(* IEC 61131-3 sources: SafeDODiag/SafeDODiag, 15 files *)

(* ---- Types.typ ---- *)
(*(Safety Release) Two-output safety contactor control and diagnosis*)
TYPE
	SContactorStateEnum :
		(
		SC_CFG := 0,
		SC_INIT,
		SC_DISABLED,
		SC_ENABLED,
		SC_ERROR := -1
		);
	SContactorCmdSimType : 	STRUCT
		EnableSim : BOOL; (*Enable contactor input and output simulation. Use fub output Simulation to see the expected output values and feedback values.*)
		SimMonitorErrors : USINT; (*Simulate error conditions by toggling individual bits to TRUE:
0: output 1 blocked by safety (interlock)
1: output 2 blocked by safety (interlock)
2: output 1 wire break (current)
3: output 2 wire break (current)
4: fdbk 1 stuck on high/"contactor open" (fdbk)
5: fdbk 2 stuck on high/"contactor open" (fdbk)
6: fdbk 1 stuck on low/"contactor closed" (fdbk)
7: fdbk 2 stuck on low/"contactor closed" (fdbk)*)
	END_STRUCT;
	SContactorCmdType : 	STRUCT
		OutputRequest : BOOL; (*Process control request: TRUE - close the contactor; FALSE - open the contactor*)
		Reset : BOOL; (*Remove the gray CPU fub from its error state and send reset request to safety CPU*)
		Simulation : SContactorCmdSimType; (*Simulation request. Element "SimMonitorErrors" only gets checked if element "EnableSim" is set to TRUE.*)
	END_STRUCT;
	SContactorCfgDiagCodeType : 	STRUCT  (*Configure safety CPU-reported SF_EDM fub DiagCode monitoring*)
		EnableMon : BOOL; (*When TRUE the contactor function block will monitor safety CPU's SF_EDM fub DiagCodes (require safety CPU to use UINT channels to pass DiagCodes to gray CPU)*)
		StartDelayTime : TIME := T#3s; (*The amount of time the gray CPU fub will delay checking SF_EDM fub DiagCode after SI card shows SafeModuleOK (must be > SF_EDM MonitorTime to allow SF_EDM to produce a stabilized DiagCode)*)
		ResetDelayTime : TIME := T#1s; (*The amount of time the gray CPU fub will delay requesting to reset SF_EDM fub after DiagCode shows 16#C060 (to allow channel diagnosis to complete and contactor feedbacks to show TRUE after SI card reports SafeModuleOK); also used as the amount of time the gray CPU fub will wait to reset itself after requesting to reset SF_EDM fub.*)
	END_STRUCT;
	SContactorCfgFdbkType : 	STRUCT  (*Configure SI hardware-based contactor status feedback monitoring*)
		EnableMon : BOOL; (*When TRUE the contactor function block will monitor SI hardware for contactor status feedback*)
		StartDelayTime : TIME := T#3s; (*The amount of time the gray CPU fub will delay checking contactor feedbacks after SI card shows SafeModuleOK (to allow channel diagnosis to complete and contactor feedbacks to show TRUE after SI card reports SafeModuleOK)*)
		MonitorTime : TIME; (*The amount of time the gray CPU fub will delay comparing contactor feedbacks to allow for switching time and debounce*)
	END_STRUCT;
	SContactorCfgCurrentType : 	STRUCT  (*Configure SO hardware-based current ok monitoring*)
		EnableMon : BOOL; (*When true the contactor function block will monitor the current input for the contactor*)
		MonitorTime : TIME; (*The amount of time the gray CPU fub will delay checking the current output to allow transient current to settle*)
	END_STRUCT;
	SContactorCfgInterlockStateType : 	STRUCT  (*Dual-channel safe digital output: Configure SO hardware-based output interlock state ("restart inhibit state") monitoring*)
		EnableMon : BOOL; (*When TRUE the contactor function block will monitor SO hardware for output interlock state (require SO card's "Restart inhibit state information" turned on)*)
		ChannelPairSelector : USINT; (*Selector for which byte of the output interlock channel represents the contactor pair (1 - contactor pair is on SO card channels 1 & 2; 3 - contactor pair is on SO card channels 3 & 4; 5 - contactor pair is on SO card channels 5 & 6; 0/2/4/etc. - selection invalid)*)
		StartDelayTime : TIME := T#3s; (*The amount of time the gray CPU fub will delay checking output interlock states after SO card shows SafeModuleOK (to allow channel diagnosis to complete after SO card reports SafeModuleOK)*)
		MonitorTime : TIME; (*The amount of time the gray CPU fub will delay comparing interlock states' discrepancy*)
	END_STRUCT;
	SContactorCfgType : 	STRUCT
		Name : STRING[35] := 'NamedContactors'; (*Unique contactor name for easy identification in alarm text*)
		DiagCode : SContactorCfgDiagCodeType; (*Option for monitoring safety CPU's SF_EDM fub state*)
		Fdbk : SContactorCfgFdbkType; (*Option for monitoring status input of each contactors*)
		Current : SContactorCfgCurrentType; (*Option for monitoring current associated with the pair of contactors*)
		InterlockState : SContactorCfgInterlockStateType; (*Option for monitoring output interlock state of each contactor*)
		BootUpDelay : TIME := T#10m; (*Wait time for the SafeModuleOK feedback on PLC startup*)
	END_STRUCT;
	SContactorSimulationType : 	STRUCT
		Input : SContactorIntInputType; (*Simulation inputs mirror the internal inputs, so the data type uses SContactorIntInputType (not a typo)*)
		Output : SContactorIntOutputType; (*Simulation inputs mirror the internal outputs, so the data type uses SContactorIntOutputType (not a typo)*)
	END_STRUCT;
	SContactorStatusType : 	STRUCT
		OutputRequested : BOOL; (*Echo the OutputRequest input to show that the fub is running*)
		OutputActive : BOOL; (*Show that both safety contactor outputs are energized (safety contactors are not necessarily closed)*)
		SafetyResetRequested : BOOL; (*Show that a SF_EDM reset needs to be sent to safety CPU*)
	END_STRUCT;
	SContactorDiagType : 	STRUCT
		DiagText : STRING[79];
		ErrorConfig : BOOL; (*The error is due to an invalid config*)
		ErrorSafeFub : BOOL; (*The error is due to safety CPU fub SF_EDM*)
		ErrorFdbk : BOOL; (*The error is due to contactor status feedback*)
		ErrorCurrent : BOOL; (*The error is due to current feedback*)
		ErrorInterlock : BOOL; (*The error is due to output interlock*)
		ErrorInternal : BOOL; (*The error is due to fub design that did not account for certain situations*)
	END_STRUCT;
	SContactorIntPrevType : 	STRUCT
		State : SContactorStateEnum;
		Reset : BOOL;
		EnDiagCode : BOOL;
		EnFdbk : BOOL;
		EnInterlock : BOOL;
		EnCurrent : BOOL;
		SimOutput1 : BOOL;
		SimOutput2 : BOOL;
	END_STRUCT;
	SContactorIntFubType : 	STRUCT
		TON_EDMStartDelay : TON;
		TON_EDMResetDelay : TON;
		TON_FdbkStartDelay : TON;
		TON_Fdbk : TON;
		TON_Current : TON;
		TON_InterlockStartDelay : TON;
		TON_Interlock : TON;
		TON_EDMMonitorSim : TON;
	END_STRUCT;
	SContactorIntInputType : 	STRUCT
		SF_In_DiagCode : UINT;
		SI_In_SafeModuleOK : BOOL;
		SI_In_Contactor1Fdbk : BOOL;
		SI_In_Contactor2Fdbk : BOOL;
		SO_In_SafeModuleOK : BOOL;
		SO_In_Output1PhysicalState : BOOL;
		SO_In_Output2PhysicalState : BOOL;
		SO_In_Output1CurrentOK : BOOL;
		SO_In_Output2CurrentOK : BOOL;
		SO_In_OutputInterlockStates : UINT;
		InterlockStateOutput1 : USINT;
		InterlockStateOutput2 : USINT;
	END_STRUCT;
	SContactorIntOutputType : 	STRUCT
		SO_Out_Contactor1 : BOOL;
		SO_Out_Contactor2 : BOOL;
	END_STRUCT;
	SContactorInternalType : 	STRUCT
		State : SContactorStateEnum; (*State of the contactor fub*)
		StateGoTo : SContactorStateEnum;
		Input : SContactorIntInputType;
		Output : SContactorIntOutputType;
		Fub : SContactorIntFubType;
		Prev : SContactorIntPrevType;
		EDMReset : BOOL;
		i : UDINT;
	END_STRUCT;
END_TYPE

(*(Safety Release) Single-channel safe digital output control and diagnosis (a simplification of SContactor)*)

TYPE
	SDigitalOutCfgInterlockStateType : 	STRUCT  (*Single-channel safe digital output: Configure SO hardware-based output interlock state ("restart inhibit state") monitoring*)
		EnableMon : BOOL; (*When TRUE the contactor function block will monitor SO hardware for output interlock state (require SO card's "Restart inhibit state information" turned on)*)
		ChannelSelector : USINT; (*Selector for which byte of the output interlock channel represents the contactor pair (1/2/3/4 for Safety Release, or 1/2 for mapp Safety - SO card channel that's being controlled; 0 or any other number - selection invalid)*)
		StartDelayTime : TIME := T#3s; (*The amount of time the gray CPU fub will delay checking output interlock states after SO card shows SafeModuleOK (to allow channel diagnosis to complete after SO card reports SafeModuleOK)*)
		MonitorTime : TIME; (*The amount of time the gray CPU fub will delay comparing interlock states' discrepancy*)
	END_STRUCT;
	SDigitalOutCfgType : 	STRUCT
		Name : STRING[35]; (*Unique contactor name for easy identification in alarm text*)
		DiagCode : SContactorCfgDiagCodeType; (*Option for monitoring safety CPU's SF_EDM fub state*)
		Fdbk : SContactorCfgFdbkType; (*Option for monitoring status input of each contactors*)
		Current : SContactorCfgCurrentType; (*Option for monitoring current associated with the pair of contactors*)
		InterlockState : SDigitalOutCfgInterlockStateType; (*Option for monitoring output interlock state of each contactor*)
	END_STRUCT;
END_TYPE

(*(mapp Safety) Interlock state monitoring for two-output safety contactor control (a modification of SContactor)*)

TYPE
	SfContactorCfgInterlockStateType : 	STRUCT  (*Dual-channel safe digital output: Configure SO hardware-based output interlock state ("error interlock state") monitoring*)
		EnableMon : BOOL; (*When TRUE the contactor function block will monitor SO hardware for output interlock state (require SO card's "Restart inhibit state information" turned on)*)
		StartDelayTime : TIME := T#3s; (*The amount of time the gray CPU fub will delay checking output interlock states after SO card shows SafeModuleOK (to allow channel diagnosis to complete after SO card reports SafeModuleOK)*)
		MonitorTime : TIME; (*The amount of time the gray CPU fub will delay comparing interlock states' discrepancy*)
	END_STRUCT;
	SfContactorCfgType : 	STRUCT
		Name : STRING[35] := 'NamedContactors'; (*Unique contactor name for easy identification in alarm text*)
		DiagCode : SContactorCfgDiagCodeType; (*Option for monitoring safety CPU's SF_EDM fub state*)
		Fdbk : SContactorCfgFdbkType; (*Option for monitoring status input of each contactors*)
		Current : SContactorCfgCurrentType; (*Option for monitoring current associated with the pair of contactors*)
		InterlockState : SfContactorCfgInterlockStateType; (*Option for monitoring output interlock state of each contactor*)
		BootUpDelay : TIME := T#10m; (*Wait time for the SafeModuleOK feedback on PLC startup*)
	END_STRUCT;
	SfContactorIntInputType : 	STRUCT
		SF_In_DiagCode : UINT;
		SI_In_SafeModuleOK : BOOL;
		SI_In_Contactor1Fdbk : BOOL;
		SI_In_Contactor2Fdbk : BOOL;
		SO_In_SafeModuleOK : BOOL;
		SO_In_Output1PhysicalState : BOOL;
		SO_In_Output2PhysicalState : BOOL;
		SO_In_Output1CurrentOK : BOOL;
		SO_In_Output2CurrentOK : BOOL;
		SO_In_OutputInterlockStates : USINT;
		InterlockStateOutput1 : USINT;
		InterlockStateOutput2 : USINT;
	END_STRUCT;
	SfContactorInternalType : 	STRUCT
		State : SContactorStateEnum; (*State of the contactor fub*)
		StateGoTo : SContactorStateEnum;
		Input : SfContactorIntInputType;
		Output : SContactorIntOutputType;
		Fub : SContactorIntFubType;
		Prev : SContactorIntPrevType;
		EDMReset : BOOL;
		i : UDINT;
	END_STRUCT;
END_TYPE

(* ---- SafeDODiag.fun ---- *)
(*Safety Release-compatible X20SO21xx/X20SO41xx output error diagnosis*)
FUNCTION_BLOCK SContactor (*Dual-channel safe digital output control and monitoring, example use includes redundant safety contactor control*)
	VAR_INPUT
		Cmd : SContactorCmdType; (*Request to energize output*)
		pSO_Out_Contactor1 : REFERENCE TO BOOL; (*Reference to the SO card output for contactor coil 1*)
		pSO_Out_Contactor2 : REFERENCE TO BOOL; (*Reference to the SO card output for contactor coil 2*)
		pSO_In_SafeModuleOK : REFERENCE TO BOOL; (*Reference to the SO card input SafeModuleOK*)
		pSO_In_Output1PhysicalState : REFERENCE TO BOOL; (*Reference to the SO card input PhysicalStateChannelX for contactor coil 1*)
		pSO_In_Output2PhysicalState : REFERENCE TO BOOL; (*Reference to the SO card input PhysicalStateChannelY for contactor coil 2*)
		Config : SContactorCfgType; (*Pointer to the configuration structure*)
		pSF_In_DiagCode : REFERENCE TO UINT; (*Reference to the safety-to-gray UINT channel that reports SF_EDM fub DiagCode*)
		pSI_In_SafeModuleOK : REFERENCE TO BOOL; (*Reference to the SO card input SafeModuleOK*)
		pSI_In_Contactor1Fdbk : REFERENCE TO BOOL; (*Reference to the SI card input for the feedback status of contactor coil 1*)
		pSI_In_Contactor2Fdbk : REFERENCE TO BOOL; (*Reference to the SI card input for the feedback status of contactor coil 2*)
		pSO_In_Output1CurrentOK : REFERENCE TO BOOL; (*Reference to the SO card's monitoring of channel current for contactor coil 1*)
		pSO_In_Output2CurrentOK : REFERENCE TO BOOL; (*Reference to the SO card's monitoring of channel current for contactor coil 2*)
		pSO_In_OutputInterlockStates : REFERENCE TO UINT; (*Reference to the SO card output interlocking states (each channel is 1 nibble in the range of 16#0 - 16#F)*)
		pSO6_In_OutputInterlockStates : REFERENCE TO UDINT; (*Reference to the SO6xxx card output interlocking states (each channel is 1 nibble in the range of 16#0 - 16#F)*)
	END_VAR
	VAR_OUTPUT
		Error : BOOL; (*Show that an error has occured to prevent output*)
		DiagCode : UINT; (*Show diagnostic code based on available monitoring capability*)
		Diag : SContactorDiagType; (*Show diagnostic info based on available monitoring capability*)
		Status : SContactorStatusType; (*Show that both safety contactor outputs are energized (safety contactors are not necessarily closed)*)
		Simulation : SContactorSimulationType; (*Show simulated I/O values based on fub input Cmd.Simulation.SimMonitorErrors*)
	END_VAR
	VAR
		Internal : SContactorInternalType; (*Internal variables*)
	END_VAR
END_FUNCTION_BLOCK

FUNCTION_BLOCK SDigitalOut (*Single-channel safe digital output control and monitoring, example use includes gas dump valve control*)
	VAR_INPUT
		Cmd : SContactorCmdType; (*Request to energize output*)
		pSO_Out_DigitalOut : REFERENCE TO BOOL; (*Reference to the SO card digital output channel*)
		pSO_In_SafeModuleOK : REFERENCE TO BOOL; (*Reference to the SO card input SafeModuleOK*)
		pSO_In_OutputPhysicalState : REFERENCE TO BOOL; (*Reference to the SO card input PhysicalStateChannelX for the controlled digital output channel*)
		Config : SDigitalOutCfgType; (*Pointer to the configuration structure*)
		pSF_In_DiagCode : REFERENCE TO UINT; (*Reference to the safety-to-gray UINT channel that reports SF_EDM fub DiagCode*)
		pSI_In_SafeModuleOK : REFERENCE TO BOOL; (*Reference to the SO card input SafeModuleOK*)
		pSI_In_DigitalOutFdbk : REFERENCE TO BOOL; (*Reference to the SI card input for the feedback status of the controlled digital output channel*)
		pSO_In_OutputCurrentOK : REFERENCE TO BOOL; (*Reference to the SO card's monitoring of channel current for the controlled digital output channel*)
		pSO_In_OutputInterlockStates : REFERENCE TO UINT; (*Reference to the SO card output interlocking states (each channel is 1 nibble in the range of 16#0 - 16#F)*)
		pSO6_In_OutputInterlockStates : REFERENCE TO UDINT; (*Reference to the SO6xxx card output interlocking states (each channel is 1 nibble in the range of 16#0 - 16#F)*)
	END_VAR
	VAR_OUTPUT
		Error : BOOL; (*Show that an error has occured to prevent output*)
		DiagCode : UINT; (*Show diagnostic code based on available monitoring capability*)
		Diag : SContactorDiagType; (*Show diagnostic info based on available monitoring capability*)
		Status : SContactorStatusType; (*Show that safety digiral output is energized*)
		Simulation : SContactorSimulationType; (*Show simulated I/O values based on fub input Cmd.Simulation.SimMonitorErrors*)
	END_VAR
	VAR
		Internal : SContactorInternalType; (*Internal variables*)
	END_VAR
END_FUNCTION_BLOCK
(*mapp Safety-compatible X20SO21xx/X20SO41xx output error diagnosis*)

FUNCTION_BLOCK SfContactor (*Dual-channel safe digital output control and monitoring, example use includes redundant safety contactor control*)
	VAR_INPUT
		Cmd : SContactorCmdType; (*Request to energize output*)
		pSO_Out_Contactor1 : REFERENCE TO BOOL; (*Reference to the SO card output for contactor coil 1*)
		pSO_Out_Contactor2 : REFERENCE TO BOOL; (*Reference to the SO card output for contactor coil 2*)
		pSO_In_SafeModuleOK : REFERENCE TO BOOL; (*Reference to the SO card input SafeModuleOK*)
		pSO_In_Output1PhysicalState : REFERENCE TO BOOL; (*Reference to the SO card input PhysicalStateChannelX for contactor coil 1*)
		pSO_In_Output2PhysicalState : REFERENCE TO BOOL; (*Reference to the SO card input PhysicalStateChannelY for contactor coil 2*)
		Config : SfContactorCfgType; (*Pointer to the configuration structure*)
		pSF_In_DiagCode : REFERENCE TO UINT; (*Reference to the safety-to-gray UINT channel that reports SF_EDM fub DiagCode*)
		pSI_In_SafeModuleOK : REFERENCE TO BOOL; (*Reference to the SO card input SafeModuleOK*)
		pSI_In_Contactor1Fdbk : REFERENCE TO BOOL; (*Reference to the SI card input for the feedback status of contactor coil 1*)
		pSI_In_Contactor2Fdbk : REFERENCE TO BOOL; (*Reference to the SI card input for the feedback status of contactor coil 2*)
		pSO_In_Output1CurrentOK : REFERENCE TO BOOL; (*Reference to the SO card's monitoring of channel current for contactor coil 1*)
		pSO_In_Output2CurrentOK : REFERENCE TO BOOL; (*Reference to the SO card's monitoring of channel current for contactor coil 2*)
		pSO_In_OutputInterlockStates : REFERENCE TO USINT; (*Reference to the SO card output interlocking states (each channel is 1 nibble in the range of 16#0 - 16#F)*)
	END_VAR
	VAR_OUTPUT
		Error : BOOL; (*Show that an error has occured to prevent output*)
		DiagCode : UINT; (*Show diagnostic code based on available monitoring capability*)
		Diag : SContactorDiagType; (*Show diagnostic info based on available monitoring capability*)
		Status : SContactorStatusType; (*Show that both safety contactor outputs are energized (safety contactors are not necessarily closed)*)
		Simulation : SContactorSimulationType; (*Show simulated I/O values based on fub input Cmd.Simulation.SimMonitorErrors*)
	END_VAR
	VAR
		Internal : SfContactorInternalType; (*Internal variables*)
	END_VAR
END_FUNCTION_BLOCK

FUNCTION_BLOCK SfDigitalOut (*Single-channel safe digital output control and monitoring, example use includes gas dump valve control*)
	VAR_INPUT
		Cmd : SContactorCmdType; (*Request to energize output*)
		pSO_Out_DigitalOut : REFERENCE TO BOOL; (*Reference to the SO card digital output channel*)
		pSO_In_SafeModuleOK : REFERENCE TO BOOL; (*Reference to the SO card input SafeModuleOK*)
		pSO_In_OutputPhysicalState : REFERENCE TO BOOL; (*Reference to the SO card input PhysicalStateChannelX for the controlled digital output channel*)
		Config : SDigitalOutCfgType; (*Pointer to the configuration structure*)
		pSF_In_DiagCode : REFERENCE TO UINT; (*Reference to the safety-to-gray UINT channel that reports SF_EDM fub DiagCode*)
		pSI_In_SafeModuleOK : REFERENCE TO BOOL; (*Reference to the SO card input SafeModuleOK*)
		pSI_In_DigitalOutFdbk : REFERENCE TO BOOL; (*Reference to the SI card input for the feedback status of the controlled digital output channel*)
		pSO_In_OutputCurrentOK : REFERENCE TO BOOL; (*Reference to the SO card's monitoring of channel current for the controlled digital output channel*)
		pSO_In_OutputInterlockStates : REFERENCE TO USINT; (*Reference to the SO card output interlocking states (each channel is 1 nibble in the range of 16#0 - 16#F)*)
	END_VAR
	VAR_OUTPUT
		Error : BOOL; (*Show that an error has occured to prevent output*)
		DiagCode : UINT; (*Show diagnostic code based on available monitoring capability*)
		Diag : SContactorDiagType; (*Show diagnostic info based on available monitoring capability*)
		Status : SContactorStatusType; (*Show that safety digiral output is energized*)
		Simulation : SContactorSimulationType; (*Show simulated I/O values based on fub input Cmd.Simulation.SimMonitorErrors*)
	END_VAR
	VAR
		Internal : SfContactorInternalType; (*Internal variables*)
	END_VAR
END_FUNCTION_BLOCK

(* ---- SContactor.st ---- *)
(*
This fub has four monitoring options, ordered by priority below:
1) SF_EDM DiagCode from safety CPU (highest priority)
2) external contactor state monitoring (using SafeDigitalInput0x from SI card)
3) internal contactor wiring monitoring (using CurrentOK0x from SO card)
4) output interlock state monitoring (using FBK_Status_1 from SO card) (lowest priority)
If more than one monitoring options are enabled, the highest priority option will be used by the fub to evaluate contactor open/close behavior.
##################################################*)

FUNCTION_BLOCK SContactor

	//########## Simulation input handling ##########
	IF ( Cmd.Simulation.EnableSim ) THEN
		Simulation.Input.SI_In_SafeModuleOK	:= TRUE;
		Simulation.Input.SO_In_SafeModuleOK	:= TRUE;

		Internal.i	:= TIME_TO_UDINT( clock_ms() ) MOD 200;

		//########## SContactor dual-channel input simulation ##########
		// SimMonitorErrors bits (when set to TRUE):
		//  0: output 1 blocked by safety (interlock)
		//  1: output 2 blocked by safety (interlock)
		//  2: output 1 wire break (current)
		//  3: output 2 wire break (current)
		//  4: fdbk 1 stuck on high/"contactor open" (fdbk)
		//  5: fdbk 2 stuck on high/"contactor open" (fdbk)
		//  6: fdbk 1 stuck on low/"contactor closed" (fdbk)
		//  7: fdbk 2 stuck on low/"contactor closed" (fdbk)

		// simulate interlock feedback
		IF ( Cmd.Simulation.SimMonitorErrors.0 ) THEN
			Simulation.Input.SO_In_Output1PhysicalState	:= FALSE;
			Simulation.Input.InterlockStateOutput1		:= 8;
		ELSE
			Simulation.Input.SO_In_Output1PhysicalState	:= Simulation.Output.SO_Out_Contactor1 AND ( Simulation.Input.SO_In_Output1PhysicalState OR ( Internal.i >= 0	AND Internal.i < 50 ) );
			IF ( Simulation.Input.SO_In_Output1PhysicalState ) THEN
				Simulation.Input.InterlockStateOutput1	:= 9;
			ELSE
				Simulation.Input.InterlockStateOutput1	:= 7;
			END_IF
		END_IF
		IF ( Cmd.Simulation.SimMonitorErrors.1 ) THEN
			Simulation.Input.SO_In_Output2PhysicalState	:= FALSE;
			Simulation.Input.InterlockStateOutput2		:= 8;
		ELSE
			Simulation.Input.SO_In_Output2PhysicalState	:= Simulation.Output.SO_Out_Contactor2 AND ( Simulation.Input.SO_In_Output2PhysicalState OR ( Internal.i >= 15	AND Internal.i < 65 ) );
			IF ( Simulation.Input.SO_In_Output2PhysicalState ) THEN
				Simulation.Input.InterlockStateOutput2	:= 9;
			ELSE
				Simulation.Input.InterlockStateOutput2	:= 7;
			END_IF
		END_IF

		// simulate current ok feedback
		IF ( Cmd.Simulation.SimMonitorErrors.2 ) THEN
			Simulation.Input.SO_In_Output1CurrentOK	:= FALSE;
		ELSE
			Simulation.Input.SO_In_Output1CurrentOK	:= Simulation.Input.SO_In_Output1PhysicalState AND ( Simulation.Input.SO_In_Output1CurrentOK OR ( Internal.i >= 30	AND Internal.i < 80 ) );
		END_IF
		IF ( Cmd.Simulation.SimMonitorErrors.3 ) THEN
			Simulation.Input.SO_In_Output2CurrentOK	:= FALSE;
		ELSE
			Simulation.Input.SO_In_Output2CurrentOK	:= Simulation.Input.SO_In_Output2PhysicalState AND ( Simulation.Input.SO_In_Output2CurrentOK OR ( Internal.i >= 45	AND Internal.i < 95 ) );
		END_IF

		// simulate external monitoring feedback
		IF ( Cmd.Simulation.SimMonitorErrors.4 ) THEN
			Simulation.Input.SI_In_Contactor1Fdbk	:= TRUE;
		ELSIF ( Cmd.Simulation.SimMonitorErrors.6 ) THEN
			Simulation.Input.SI_In_Contactor1Fdbk	:= FALSE;
		ELSE
			IF ( Internal.i >= 60 AND Internal.i < 110 ) THEN
				IF ( Simulation.Input.SO_In_Output1CurrentOK ) THEN
					Simulation.Input.SI_In_Contactor1Fdbk	:= FALSE;
				ELSE
					Simulation.Input.SI_In_Contactor1Fdbk	:= TRUE;
				END_IF
			END_IF
		END_IF
		IF ( Cmd.Simulation.SimMonitorErrors.5 ) THEN
			Simulation.Input.SI_In_Contactor2Fdbk	:= TRUE;
		ELSIF ( Cmd.Simulation.SimMonitorErrors.7 ) THEN
			Simulation.Input.SI_In_Contactor2Fdbk	:= FALSE;
		ELSE
			IF ( Internal.i >= 75 AND Internal.i < 125 ) THEN
				IF ( Simulation.Input.SO_In_Output2CurrentOK ) THEN
					Simulation.Input.SI_In_Contactor2Fdbk	:= FALSE;
				ELSE
					Simulation.Input.SI_In_Contactor2Fdbk	:= TRUE;
				END_IF
			END_IF
		END_IF

		//########## DiagCode simulation ##########
		SimAction_DiagCode;

		//########## SContactor dual-channel input source assignment ##########
		Internal.Input.SF_In_DiagCode		:= Simulation.Input.SF_In_DiagCode;
		Internal.Input.SI_In_SafeModuleOK		:= Simulation.Input.SI_In_SafeModuleOK;
		Internal.Input.SI_In_Contactor1Fdbk		:= Simulation.Input.SI_In_Contactor1Fdbk;
		Internal.Input.SI_In_Contactor2Fdbk		:= Simulation.Input.SI_In_Contactor2Fdbk;
		Internal.Input.SO_In_SafeModuleOK			:= Simulation.Input.SO_In_SafeModuleOK;
		Internal.Input.SO_In_Output1PhysicalState	:= Simulation.Input.SO_In_Output1PhysicalState;
		Internal.Input.SO_In_Output2PhysicalState	:= Simulation.Input.SO_In_Output2PhysicalState;
		Internal.Input.SO_In_Output1CurrentOK		:= Simulation.Input.SO_In_Output1CurrentOK;
		Internal.Input.SO_In_Output2CurrentOK		:= Simulation.Input.SO_In_Output2CurrentOK;
		IF ( Config.InterlockState.ChannelPairSelector = 1 ) THEN
			Internal.Input.SO_In_OutputInterlockStates	:= Simulation.Input.InterlockStateOutput1 + Simulation.Input.InterlockStateOutput2 * 16#10;
		ELSIF ( Config.InterlockState.ChannelPairSelector = 3 ) THEN
			Internal.Input.SO_In_OutputInterlockStates	:= Simulation.Input.InterlockStateOutput1 * 16#100 + Simulation.Input.InterlockStateOutput2 * 16#1000;
		ELSIF ( Config.InterlockState.ChannelPairSelector = 5 AND ADR(pSO6_In_OutputInterlockStates) > 0 ) THEN
			Internal.Input.SO_In_OutputInterlockStates	:= Simulation.Input.InterlockStateOutput1 * 16#10000 + Simulation.Input.InterlockStateOutput2 * 16#100000;
		ELSE
			Internal.Input.SO_In_OutputInterlockStates	:= 0;
		END_IF

	ELSE
		//########## SContactor dual-channel input source assignment ##########
		IF ( ADR(pSF_In_DiagCode) > 0 ) THEN
			Internal.Input.SF_In_DiagCode		:= pSF_In_DiagCode;
		ELSE
			Internal.Input.SF_In_DiagCode		:= 0;
		END_IF
		IF ( ADR(pSI_In_SafeModuleOK) > 0 ) THEN
			Internal.Input.SI_In_SafeModuleOK	:= pSI_In_SafeModuleOK;
		ELSE
			Internal.Input.SI_In_SafeModuleOK	:= 0;
		END_IF
		IF ( ADR(pSI_In_Contactor1Fdbk) > 0 ) THEN
			Internal.Input.SI_In_Contactor1Fdbk	:= pSI_In_Contactor1Fdbk;
		ELSE
			Internal.Input.SI_In_Contactor1Fdbk	:= 0;
		END_IF
		IF ( ADR(pSI_In_Contactor2Fdbk) > 0 ) THEN
			Internal.Input.SI_In_Contactor2Fdbk	:= pSI_In_Contactor2Fdbk;
		ELSE
			Internal.Input.SI_In_Contactor2Fdbk	:= 0;
		END_IF
		IF ( ADR(pSO_In_SafeModuleOK) > 0 ) THEN
			Internal.Input.SO_In_SafeModuleOK			:= pSO_In_SafeModuleOK;
		ELSE
			Internal.Input.SO_In_SafeModuleOK			:= 0;
		END_IF
		IF ( ADR(pSO_In_Output1PhysicalState) > 0 ) THEN
			Internal.Input.SO_In_Output1PhysicalState	:= pSO_In_Output1PhysicalState;
		ELSE
			Internal.Input.SO_In_Output1PhysicalState	:= 0;
		END_IF
		IF ( ADR(pSO_In_Output2PhysicalState) > 0 ) THEN
			Internal.Input.SO_In_Output2PhysicalState	:= pSO_In_Output2PhysicalState;
		ELSE
			Internal.Input.SO_In_Output2PhysicalState	:= 0;
		END_IF
		IF ( ADR(pSO_In_Output1CurrentOK) > 0 ) THEN
			Internal.Input.SO_In_Output1CurrentOK		:= pSO_In_Output1CurrentOK;
		ELSE
			Internal.Input.SO_In_Output1CurrentOK		:= 0;
		END_IF
		IF ( ADR(pSO_In_Output2CurrentOK) > 0 ) THEN
			Internal.Input.SO_In_Output2CurrentOK		:= pSO_In_Output2CurrentOK;
		ELSE
			Internal.Input.SO_In_Output2CurrentOK		:= 0;
		END_IF
		IF ( ADR(pSO6_In_OutputInterlockStates) > 0 ) THEN
			Internal.Input.SO_In_OutputInterlockStates	:= pSO6_In_OutputInterlockStates;
		ELSIF ( ADR(pSO_In_OutputInterlockStates) > 0 ) THEN
			Internal.Input.SO_In_OutputInterlockStates	:= UINT_TO_UDINT( pSO_In_OutputInterlockStates );
		ELSE
			Internal.Input.SO_In_OutputInterlockStates	:= 0;
		END_IF
		//########## Reset simulation inputs ##########
		brsmemset( ADR(Simulation.Input), 0, SIZEOF(Simulation.Input) );

	END_IF

	//########## SContactor dual-channel output interlock state identification ##########
	// Read output channel interlock state
	IF ( Config.InterlockState.EnableMon ) THEN
		CASE Config.InterlockState.ChannelPairSelector OF
			1:
				Internal.Input.InterlockStateOutput1 := UDINT_TO_USINT( Internal.Input.SO_In_OutputInterlockStates AND 16#00000F );
				Internal.Input.InterlockStateOutput2 := UDINT_TO_USINT( SHR(( Internal.Input.SO_In_OutputInterlockStates AND 16#0000F0 ), 4) );
			3:
				Internal.Input.InterlockStateOutput1 := UDINT_TO_USINT( SHR(( Internal.Input.SO_In_OutputInterlockStates AND 16#000F00 ), 8) );
				Internal.Input.InterlockStateOutput2 := UDINT_TO_USINT( SHR(( Internal.Input.SO_In_OutputInterlockStates AND 16#00F000 ), 12) );
			5:
				IF ( ADR(pSO6_In_OutputInterlockStates) > 0 ) THEN
					Internal.Input.InterlockStateOutput1 := UDINT_TO_USINT( SHR(( Internal.Input.SO_In_OutputInterlockStates AND 16#0F0000 ), 16) );
					Internal.Input.InterlockStateOutput2 := UDINT_TO_USINT( SHR(( Internal.Input.SO_In_OutputInterlockStates AND 16#F00000 ), 20) );
				ELSE
					Internal.Input.InterlockStateOutput1 := 0;
					Internal.Input.InterlockStateOutput2 := 0;
				END_IF
			ELSE
				Internal.Input.InterlockStateOutput1 := 0;
				Internal.Input.InterlockStateOutput2 := 0;
		END_CASE
	ELSE
		Internal.Input.InterlockStateOutput1 := 0;
		Internal.Input.InterlockStateOutput2 := 0;
	END_IF

	//########## Feedback interpretation and error state transition ##########
	StateAction_CommonPre;

	//########## State machine for processing feedback values ##########
	CASE Internal.State OF

		SC_CFG:
			//#################### Req. Checkout ####################
			IF ( ADR(pSO_In_SafeModuleOK) = 0 ) THEN // Check if the monitoring of safe communication to SO node exists
				DiagCode			:= 16#F001;
				Diag.ErrorConfig	:= TRUE;
				Diag.DiagText		:= 'NoSafeDOCardOkADR';
			ELSIF ( ADR(pSO_Out_Contactor1) = 0 ) THEN // Check if output channe l exists
				DiagCode			:= 16#F002;
				Diag.ErrorConfig	:= TRUE;
				Diag.DiagText		:= 'NoContactor1OutADR';
			ELSIF ( ADR(pSO_Out_Contactor2) = 0 ) THEN // Check if output channe 2 exists
				DiagCode			:= 16#F003;
				Diag.ErrorConfig	:= TRUE;
				Diag.DiagText		:= 'NoContactor2OutADR';
			ELSIF ( ADR(pSO_In_Output1PhysicalState) = 0 ) THEN // Check if the output phsical state monitoring exists
				DiagCode			:= 16#F004;
				Diag.ErrorConfig	:= TRUE;
				Diag.DiagText		:= 'NoOutput1PhysicalStateADR';
			ELSIF ( ADR(pSO_In_Output2PhysicalState) = 0 ) THEN // Check if the output phsical state monitoring exists
				DiagCode			:= 16#F005;
				Diag.ErrorConfig	:= TRUE;
				Diag.DiagText		:= 'NoOutput2PhysicalStateADR';
			END_IF
			// No MonitorTime for PhysicalState because we don't know when the safety CPU will approve output enable request

			//#################### Check the setup of safety-to-gray comm of SF_EDM fub DiagCode monitor ##################
			IF ( Config.DiagCode.EnableMon AND NOT(Diag.ErrorConfig) ) THEN
				IF ( ADR(pSF_In_DiagCode) = 0 ) THEN // Check if the monitoring of DiagCode from safety CPU exists
					DiagCode			:= 16#F010;
					Diag.ErrorConfig	:= TRUE;
					Diag.DiagText		:= 'NoDiagCodeADR';
				ELSIF ( ADR(pSI_In_SafeModuleOK) = 0 ) THEN // Check if the monitoring of safe communication to SI node exists
					DiagCode			:= 16#F011;
					Diag.ErrorConfig	:= TRUE;
					Diag.DiagText		:= 'NoSafeDICardOkADR';
				ELSIF ( ADR(pSI_In_Contactor1Fdbk) = 0 ) THEN // Need an SI card input to monitor
					DiagCode			:= 16#F012;
					Diag.ErrorConfig	:= TRUE;
					Diag.DiagText		:= 'NoContactor1FdbkADR';
				ELSIF ( ADR(pSI_In_Contactor2Fdbk) = 0 ) THEN // Need an SI card input to monitor
					DiagCode			:= 16#F013;
					Diag.ErrorConfig	:= TRUE;
					Diag.DiagText		:= 'NoContactor2FdbkADR';
				ELSIF ( Config.DiagCode.StartDelayTime = 0 ) THEN // Check time range
					DiagCode			:= 16#F020;
					Diag.ErrorConfig	:= TRUE;
					Diag.DiagText		:= 'NoStartDelay';
				ELSIF ( Config.DiagCode.StartDelayTime > T#2m ) THEN // Check time range
					DiagCode			:= 16#F021;
					Diag.ErrorConfig	:= TRUE;
					Diag.DiagText		:= 'StartDelayTooLong';
				ELSIF ( Config.DiagCode.ResetDelayTime = 0 ) THEN // Check time range
					DiagCode			:= 16#F022;
					Diag.ErrorConfig	:= TRUE;
					Diag.DiagText		:= 'NoResetDelay';
				ELSIF ( Config.DiagCode.ResetDelayTime > T#10s ) THEN // Check time range
					DiagCode			:= 16#F023;
					Diag.ErrorConfig	:= TRUE;
					Diag.DiagText		:= 'ResetDelayTooLong';
				END_IF

			//#################### Check the setup of Contactor Feedback monitor ####################
			ELSIF ( Config.Fdbk.EnableMon AND NOT(Diag.ErrorConfig) ) THEN
				IF ( ADR(pSI_In_SafeModuleOK) = 0 ) THEN // Check if the monitoring of safe communication to SI node exists
					DiagCode			:= 16#F011;
					Diag.ErrorConfig	:= TRUE;
					Diag.DiagText		:= 'NoSafeDICardOkADR';
				ELSIF ( ADR(pSI_In_Contactor1Fdbk) = 0 ) THEN // Need an SI card input to monitor
					DiagCode			:= 16#F012;
					Diag.ErrorConfig	:= TRUE;
					Diag.DiagText		:= 'NoContactor1FdbkADR';
				ELSIF ( ADR(pSI_In_Contactor2Fdbk) = 0 ) THEN // Need an SI card input to monitor
					DiagCode			:= 16#F013;
					Diag.ErrorConfig	:= TRUE;
					Diag.DiagText		:= 'NoContactor2FdbkADR';
				ELSIF ( Config.Fdbk.StartDelayTime = 0 ) THEN // Check time range
					DiagCode			:= 16#F020;
					Diag.ErrorConfig	:= TRUE;
					Diag.DiagText		:= 'NoStartDelay';
				ELSIF ( Config.Fdbk.StartDelayTime > T#10s ) THEN // Check time range
					DiagCode			:= 16#F021;
					Diag.ErrorConfig	:= TRUE;
					Diag.DiagText		:= 'StartDelayTooLong';
				ELSIF ( Config.Fdbk.MonitorTime = 0 ) THEN // Check time range
					DiagCode			:= 16#F024;
					Diag.ErrorConfig	:= TRUE;
					Diag.DiagText		:= 'NoMonitorTime';
				ELSIF ( Config.Fdbk.MonitorTime > T#2s ) THEN // Check time range
					DiagCode			:= 16#F025;
					Diag.ErrorConfig	:= TRUE;
					Diag.DiagText		:= 'MonitorTimeTooLong';
				END_IF

			//#################### Check the setup of Output Current monitor ##################
			ELSIF ( Config.Current.EnableMon AND NOT(Diag.ErrorConfig) ) THEN
				IF ( ADR(pSO_In_Output1CurrentOK) = 0 ) THEN
					DiagCode			:= 16#F014;
					Diag.ErrorConfig	:= TRUE;
					Diag.DiagText		:= 'NoOutput1CurrentOkADR';
				ELSIF ( ADR(pSO_In_Output2CurrentOK) = 0 ) THEN
					DiagCode			:= 16#F015;
					Diag.ErrorConfig	:= TRUE;
					Diag.DiagText		:= 'NoOutput2CurrentOkADR';
				ELSIF ( Config.Current.MonitorTime = 0 ) THEN // Check time range
					DiagCode			:= 16#F024;
					Diag.ErrorConfig	:= TRUE;
					Diag.DiagText		:= 'NoMonitorTime';
				ELSIF ( Config.Current.MonitorTime > T#2s ) THEN // Check time range
					DiagCode			:= 16#F025;
					Diag.ErrorConfig	:= TRUE;
					Diag.DiagText		:= 'MonitorTimeTooLong';
				END_IF

			//#################### Check the setup of Output Interlock monitor ##################
			ELSIF ( Config.InterlockState.EnableMon AND NOT(Diag.ErrorConfig) ) THEN
				IF ( ( ADR(pSO_In_OutputInterlockStates) = 0 AND ADR(pSO6_In_OutputInterlockStates) = 0 )
					OR ( Config.InterlockState.ChannelPairSelector = 5 AND ADR(pSO6_In_OutputInterlockStates) = 0 )
					) THEN
					DiagCode			:= 16#F016;
					Diag.ErrorConfig	:= TRUE;
					Diag.DiagText		:= 'NoOutputInterlockStateADR';
				ELSIF ( Config.InterlockState.MonitorTime = 0 ) THEN // Check time range
					DiagCode			:= 16#F024;
					Diag.ErrorConfig	:= TRUE;
					Diag.DiagText		:= 'NoMonitorTime';
				ELSIF ( Config.InterlockState.MonitorTime > T#1s ) THEN // Check time range
					DiagCode			:= 16#F025;
					Diag.ErrorConfig	:= TRUE;
					Diag.DiagText		:= 'MonitorTimeTooLong';
				ELSIF ( (Config.InterlockState.ChannelPairSelector <> 1)
					AND (Config.InterlockState.ChannelPairSelector <> 3)
					AND (Config.InterlockState.ChannelPairSelector <> 5)
					) THEN
					DiagCode			:= 16#F026;
					Diag.ErrorConfig	:= TRUE;
					Diag.DiagText		:= 'InvalidOutputInterlockChannelPairSelector';
				END_IF
			END_IF

			//#################### SUCCESS!!! ##################
			IF NOT( Diag.ErrorConfig ) THEN
				Internal.StateGoTo	:= SC_INIT;
			END_IF

		SC_INIT:
			StateAction_Init;

		SC_DISABLED:
			StateAction_Disabled;

		SC_ENABLED:
			StateAction_Enabled;

		SC_ERROR:
			StateAction_Error;

		ELSE
			//The code should not end uzp here. Report the error as unknown.
			Diag.ErrorInternal	:= TRUE;
			DiagCode			:= 16#CFFF;
			Diag.DiagText		:= 'UndocumentedError';

	END_CASE

	//########## Update fub outputs ##########
	// Update fub error output
	Error := Diag.ErrorSafeFub OR Diag.ErrorInterlock OR Diag.ErrorCurrent OR Diag.ErrorFdbk OR Diag.ErrorConfig OR Diag.ErrorInternal;

	// Update fub IO status outputs
	IF ( Internal.State > SC_INIT ) THEN
		// Update IOSP outputs after fub init is successful, so all safety outputs are in a safe state before energizing and monitoring
		Internal.Output.SO_Out_Contactor1	:= Cmd.OutputRequest;
		Internal.Output.SO_Out_Contactor2	:= Cmd.OutputRequest;

		// Update fub status outputs based on IOSP dual-channel agreement
		Status.OutputActive		:= Internal.Input.SO_In_Output1PhysicalState AND Internal.Input.SO_In_Output2PhysicalState; // both channels need to activate to energize, so all dual-channel diagreements are treated as inactive
		Status.OutputRequested	:= Internal.Output.SO_Out_Contactor1 AND Internal.Output.SO_Out_Contactor2; // both channels need to activate to energize, so all dual-channel diagreements are treated as no request
	ELSE
		// disable IOSP output during CFG state or ERROR state
		Internal.Output.SO_Out_Contactor1	:= FALSE;
		Internal.Output.SO_Out_Contactor2	:= FALSE;

		// Update fub status output based on available SContactor dual-channel IOSP data
		IF ( ADR(pSO_In_Output1PhysicalState) > 0 AND ADR(pSO_In_Output2PhysicalState) > 0 ) THEN
			Status.OutputActive	:= Internal.Input.SO_In_Output1PhysicalState AND Internal.Input.SO_In_Output2PhysicalState;
		ELSIF ( ADR(pSO_In_Output1PhysicalState) > 0 ) THEN
			Status.OutputActive	:= Internal.Input.SO_In_Output1PhysicalState;
		ELSIF ( ADR(pSO_In_Output2PhysicalState) > 0 ) THEN
			Status.OutputActive	:= Internal.Input.SO_In_Output2PhysicalState;
		ELSE
			Status.OutputActive	:= FALSE;
		END_IF
		Status.OutputRequested	:= FALSE;
	END_IF

	// Disable internal EDM reset request after a jump out of init state that's not made within the state machine (presumably into error state)
	// Note: Error state sets internal EDM reset request on rising edge of error acknowledgement, so error state needs to disable EDM reset on its own
	IF ( Internal.Prev.State = SC_INIT AND Internal.State <> SC_INIT ) THEN
		Internal.EDMReset	:= FALSE;
	END_IF
	// Pass through safety reset request in all fub states
	Status.SafetyResetRequested	:= Cmd.Reset OR Internal.EDMReset;

	//########## SContactor dual-channel Simulation output handling ##########
	IF ( Cmd.Simulation.EnableSim ) THEN
		//########## Output destination assignment ##########
		Simulation.Output.SO_Out_Contactor1	:= Internal.Output.SO_Out_Contactor1;
		Simulation.Output.SO_Out_Contactor2	:= Internal.Output.SO_Out_Contactor2;
		//########## Reset real outputs ##########
		IF ( ADR(pSO_Out_Contactor1) > 0 ) THEN
			pSO_Out_Contactor1	:= FALSE;
		END_IF
		IF ( ADR(pSO_Out_Contactor2) > 0 ) THEN
			pSO_Out_Contactor2	:= FALSE;
		END_IF
	ELSE
		//########## Output destination assignment ##########
		IF ( ADR(pSO_Out_Contactor1) > 0 ) THEN
			pSO_Out_Contactor1	:= Internal.Output.SO_Out_Contactor1;
		END_IF
		IF ( ADR(pSO_Out_Contactor2) > 0 ) THEN
			pSO_Out_Contactor2	:= Internal.Output.SO_Out_Contactor2;
		END_IF
		//########## Reset simulation outputs ##########
		Simulation.Output.SO_Out_Contactor1	:= FALSE;
		Simulation.Output.SO_Out_Contactor2	:= FALSE;
	END_IF

	//########## Update internal process ##########
	StateAction_CommmonAft;

END_FUNCTION_BLOCK

(* ---- SDigitalOut.st ---- *)
(*
This fub has four monitoring options, ordered by priority below:
1) SF_EDM DiagCode from safety CPU (highest priority)
2) external contactor state monitoring (using SafeDigitalInput0x from SI card)
3) internal contactor wiring monitoring (using CurrentOK0x from SO card)
4) output interlock state monitoring (using FBK_Status_1 from SO card) (lowest priority)
If more than one monitoring options are enabled, the highest priority option will be used by the fub to evaluate contactor open/close behavior.
##################################################*)

FUNCTION_BLOCK SDigitalOut

	//########## Simulation input handling ##########
	IF ( Cmd.Simulation.EnableSim ) THEN
		Simulation.Input.SI_In_SafeModuleOK	:= TRUE;
		Simulation.Input.SO_In_SafeModuleOK	:= TRUE;

		Internal.i	:= TIME_TO_UDINT( clock_ms() ) MOD 200;

		//########## SDigitalOut single-channel input simulation ##########
		// SimMonitorErrors bits (when set to TRUE):
		//  0: output X blocked by safety (interlock)
		//  1: output X blocked by safety (interlock)
		//  2: output X wire break (current)
		//  3: output X wire break (current)
		//  4: fdbk X stuck on high/"contactor open" (fdbk)
		//  5: fdbk X stuck on high/"contactor open" (fdbk)
		//  6: fdbk X stuck on low/"contactor closed" (fdbk)
		//  7: fdbk X stuck on low/"contactor closed" (fdbk)

		// simulate interlock feedback
		IF ( Cmd.Simulation.SimMonitorErrors.0 OR Cmd.Simulation.SimMonitorErrors.1 ) THEN
			Simulation.Input.SO_In_Output1PhysicalState	:= FALSE;
			Simulation.Input.InterlockStateOutput1		:= 8;
		ELSE
			Simulation.Input.SO_In_Output1PhysicalState	:= Simulation.Output.SO_Out_Contactor1 AND ( Simulation.Input.SO_In_Output1PhysicalState OR ( Internal.i >= 0	AND Internal.i < 50 ) );
			IF ( Simulation.Input.SO_In_Output1PhysicalState ) THEN
				Simulation.Input.InterlockStateOutput1	:= 9;
			ELSE
				Simulation.Input.InterlockStateOutput1	:= 7;
			END_IF
		END_IF

		// simulate current ok feedback
		IF ( Cmd.Simulation.SimMonitorErrors.2 OR Cmd.Simulation.SimMonitorErrors.3 ) THEN
			Simulation.Input.SO_In_Output1CurrentOK	:= FALSE;
		ELSE
			Simulation.Input.SO_In_Output1CurrentOK	:= Simulation.Input.SO_In_Output1PhysicalState AND ( Simulation.Input.SO_In_Output1CurrentOK OR ( Internal.i >= 30	AND Internal.i < 80 ) );
		END_IF

		// simulate external monitoring feedback
		IF ( Cmd.Simulation.SimMonitorErrors.4 OR Cmd.Simulation.SimMonitorErrors.5 ) THEN
			Simulation.Input.SI_In_Contactor1Fdbk	:= TRUE;
		ELSIF ( Cmd.Simulation.SimMonitorErrors.6 OR Cmd.Simulation.SimMonitorErrors.7 ) THEN
			Simulation.Input.SI_In_Contactor1Fdbk	:= FALSE;
		ELSE
			IF ( Internal.i >= 60 AND Internal.i < 110 ) THEN
				IF ( Simulation.Input.SO_In_Output1CurrentOK ) THEN
					Simulation.Input.SI_In_Contactor1Fdbk	:= FALSE;
				ELSE
					Simulation.Input.SI_In_Contactor1Fdbk	:= TRUE;
				END_IF
			END_IF
		END_IF
		Simulation.Input.SI_In_Contactor2Fdbk		:= Simulation.Input.SI_In_Contactor1Fdbk;
		Simulation.Input.SO_In_Output2PhysicalState	:= Simulation.Input.SO_In_Output1PhysicalState;
		Simulation.Input.SO_In_Output2CurrentOK		:= Simulation.Input.SO_In_Output1CurrentOK;
		Simulation.Input.InterlockStateOutput2		:= Simulation.Input.InterlockStateOutput1;

		//########## DiagCode simulation ##########
		SimAction_DiagCode;

		//########## SDigitalOut single-channel input source assignment ##########
		Internal.Input.SF_In_DiagCode		:= Simulation.Input.SF_In_DiagCode;
		Internal.Input.SI_In_SafeModuleOK		:= Simulation.Input.SI_In_SafeModuleOK;
		Internal.Input.SI_In_Contactor1Fdbk		:= Simulation.Input.SI_In_Contactor1Fdbk;
		Internal.Input.SI_In_Contactor2Fdbk		:= Simulation.Input.SI_In_Contactor2Fdbk;
		Internal.Input.SO_In_SafeModuleOK			:= Simulation.Input.SO_In_SafeModuleOK;
		Internal.Input.SO_In_Output1PhysicalState	:= Simulation.Input.SO_In_Output1PhysicalState;
		Internal.Input.SO_In_Output2PhysicalState	:= Simulation.Input.SO_In_Output2PhysicalState;
		Internal.Input.SO_In_Output1CurrentOK		:= Simulation.Input.SO_In_Output1CurrentOK;
		Internal.Input.SO_In_Output2CurrentOK		:= Simulation.Input.SO_In_Output2CurrentOK;
		CASE Config.InterlockState.ChannelSelector OF
			1:
				Internal.Input.SO_In_OutputInterlockStates	:= Simulation.Input.InterlockStateOutput1;
			2:
				Internal.Input.SO_In_OutputInterlockStates	:= Simulation.Input.InterlockStateOutput1 * 16#10;
			3:
				Internal.Input.SO_In_OutputInterlockStates	:= Simulation.Input.InterlockStateOutput1 * 16#100;
			4:
				Internal.Input.SO_In_OutputInterlockStates	:= Simulation.Input.InterlockStateOutput1 * 16#1000;
			ELSE
				Internal.Input.SO_In_OutputInterlockStates	:= 0;
		END_CASE

	ELSE
		//########## SDigitalOut single-channel input source assignment ##########
		IF ( ADR(pSF_In_DiagCode) > 0 ) THEN
			Internal.Input.SF_In_DiagCode		:= pSF_In_DiagCode;
		ELSE
			Internal.Input.SF_In_DiagCode		:= 0;
		END_IF
		IF ( ADR(pSI_In_SafeModuleOK) > 0 ) THEN
			Internal.Input.SI_In_SafeModuleOK	:= pSI_In_SafeModuleOK;
		ELSE
			Internal.Input.SI_In_SafeModuleOK	:= 0;
		END_IF
		IF ( ADR(pSI_In_DigitalOutFdbk) > 0 ) THEN
			Internal.Input.SI_In_Contactor1Fdbk	:= pSI_In_DigitalOutFdbk;
		ELSE
			Internal.Input.SI_In_Contactor1Fdbk	:= 0;
		END_IF
		IF ( ADR(pSO_In_SafeModuleOK) > 0 ) THEN
			Internal.Input.SO_In_SafeModuleOK			:= pSO_In_SafeModuleOK;
		ELSE
			Internal.Input.SO_In_SafeModuleOK			:= 0;
		END_IF
		IF ( ADR(pSO_In_OutputPhysicalState) > 0 ) THEN
			Internal.Input.SO_In_Output1PhysicalState	:= pSO_In_OutputPhysicalState;
		ELSE
			Internal.Input.SO_In_Output1PhysicalState	:= 0;
		END_IF
		IF ( ADR(pSO_In_OutputCurrentOK) > 0 ) THEN
			Internal.Input.SO_In_Output1CurrentOK		:= pSO_In_OutputCurrentOK;
		ELSE
			Internal.Input.SO_In_Output1CurrentOK		:= 0;
		END_IF
		IF ( ADR(pSO_In_OutputInterlockStates) > 0 ) THEN
			Internal.Input.SO_In_OutputInterlockStates	:= pSO_In_OutputInterlockStates;
		ELSE
			Internal.Input.SO_In_OutputInterlockStates	:= 0;
		END_IF
		Internal.Input.SI_In_Contactor2Fdbk			:= Internal.Input.SI_In_Contactor1Fdbk;
		Internal.Input.SO_In_Output2PhysicalState	:= Internal.Input.SO_In_Output1PhysicalState;
		Internal.Input.SO_In_Output2CurrentOK		:= Internal.Input.SO_In_Output1CurrentOK;
		//########## Reset simulation inputs ##########
		brsmemset( ADR(Simulation.Input), 0, SIZEOF(Simulation.Input) );

	END_IF

	//########## SDigitalOut single-channel output interlock state identification ##########
	// Read output channel interlock state
	IF ( Config.InterlockState.EnableMon ) THEN
		CASE Config.InterlockState.ChannelSelector OF
			1:
				Internal.Input.InterlockStateOutput1 := UINT_TO_USINT( Internal.Input.SO_In_OutputInterlockStates AND 16#000F );
			2:
				Internal.Input.InterlockStateOutput1 := UINT_TO_USINT( SHR(( Internal.Input.SO_In_OutputInterlockStates AND 16#00F0 ), 4) );
			3:
				Internal.Input.InterlockStateOutput1 := UINT_TO_USINT( SHR(( Internal.Input.SO_In_OutputInterlockStates AND 16#0F00 ), 8) );
			4:
				Internal.Input.InterlockStateOutput1 := UINT_TO_USINT( SHR(( Internal.Input.SO_In_OutputInterlockStates AND 16#F000 ), 12) );
			ELSE
				Internal.Input.InterlockStateOutput1 := 0;
		END_CASE
	ELSE
		Internal.Input.InterlockStateOutput1 := 0;
	END_IF
	Internal.Input.InterlockStateOutput2 := Internal.Input.InterlockStateOutput1;

	//########## Feedback interpretation and error state transition ##########
	StateAction_CommonPre;

	//########## State machine for processing feedback values ##########
	CASE Internal.State OF

		SC_CFG:
			//#################### Req. Checkout ####################
			IF ( ADR(pSO_In_SafeModuleOK) = 0 ) THEN // Check if the monitoring of safe communication to SO node exists
				DiagCode			:= 16#F001;
				Diag.ErrorConfig	:= TRUE;
				Diag.DiagText		:= 'NoSafeDOCardOkADR';
			ELSIF ( ADR(pSO_Out_DigitalOut) = 0 ) THEN // Check if output channel exists
				DiagCode			:= 16#F002;
				Diag.ErrorConfig	:= TRUE;
				Diag.DiagText		:= 'NoSafeDigitalOutADR';
			ELSIF ( ADR(pSO_In_OutputPhysicalState) = 0 ) THEN // Check if the output phsical state monitoring exists
				DiagCode			:= 16#F004;
				Diag.ErrorConfig	:= TRUE;
				Diag.DiagText		:= 'NoOutputPhysicalStateADR';
			END_IF
			// No MonitorTime for PhysicalState because we don't know when the safety CPU will approve output enable request

			//#################### Check the setup of safety-to-gray comm of SF_EDM fub DiagCode monitor ##################
			IF ( Config.DiagCode.EnableMon AND NOT(Diag.ErrorConfig) ) THEN
				IF ( ADR(pSF_In_DiagCode) = 0 ) THEN // Check if the monitoring of DiagCode from safety CPU exists
					DiagCode			:= 16#F010;
					Diag.ErrorConfig	:= TRUE;
					Diag.DiagText		:= 'NoDiagCodeADR';
				ELSIF ( ADR(pSI_In_SafeModuleOK) = 0 ) THEN // Check if the monitoring of safe communication to SI node exists
					DiagCode			:= 16#F011;
					Diag.ErrorConfig	:= TRUE;
					Diag.DiagText		:= 'NoSafeDICardOkADR';
				ELSIF ( ADR(pSI_In_DigitalOutFdbk) = 0 ) THEN // Need an SI card input to monitor
					DiagCode			:= 16#F012;
					Diag.ErrorConfig	:= TRUE;
					Diag.DiagText		:= 'NoDigitalOutFdbkADR';
				ELSIF ( Config.DiagCode.StartDelayTime = 0 ) THEN // Check time range
					DiagCode			:= 16#F020;
					Diag.ErrorConfig	:= TRUE;
					Diag.DiagText		:= 'NoStartDelay';
				ELSIF ( Config.DiagCode.StartDelayTime > T#10s ) THEN // Check time range
					DiagCode			:= 16#F021;
					Diag.ErrorConfig	:= TRUE;
					Diag.DiagText		:= 'StartDelayTooLong';
				ELSIF ( Config.DiagCode.ResetDelayTime = 0 ) THEN // Check time range
					DiagCode			:= 16#F022;
					Diag.ErrorConfig	:= TRUE;
					Diag.DiagText		:= 'NoResetDelay';
				ELSIF ( Config.DiagCode.ResetDelayTime > T#10s ) THEN // Check time range
					DiagCode			:= 16#F023;
					Diag.ErrorConfig	:= TRUE;
					Diag.DiagText		:= 'ResetDelayTooLong';
				END_IF

			//#################### Check the setup of Contactor Feedback monitor ####################
			ELSIF ( Config.Fdbk.EnableMon AND NOT(Diag.ErrorConfig) ) THEN
				IF ( ADR(pSI_In_SafeModuleOK) = 0 ) THEN // Check if the monitoring of safe communication to SI node exists
					DiagCode			:= 16#F011;
					Diag.ErrorConfig	:= TRUE;
					Diag.DiagText		:= 'NoSafeDICardOkADR';
				ELSIF ( ADR(pSI_In_DigitalOutFdbk) = 0 ) THEN // Need an SI card input to monitor
					DiagCode			:= 16#F012;
					Diag.ErrorConfig	:= TRUE;
					Diag.DiagText		:= 'NoDigitalOutFdbkADR';
				ELSIF ( Config.Fdbk.StartDelayTime = 0 ) THEN // Check time range
					DiagCode			:= 16#F020;
					Diag.ErrorConfig	:= TRUE;
					Diag.DiagText		:= 'NoStartDelay';
				ELSIF ( Config.Fdbk.StartDelayTime > T#10s ) THEN // Check time range
					DiagCode			:= 16#F021;
					Diag.ErrorConfig	:= TRUE;
					Diag.DiagText		:= 'StartDelayTooLong';
				ELSIF ( Config.Fdbk.MonitorTime = 0 ) THEN // Check time range
					DiagCode			:= 16#F024;
					Diag.ErrorConfig	:= TRUE;
					Diag.DiagText		:= 'NoMonitorTime';
				ELSIF ( Config.Fdbk.MonitorTime > T#2s ) THEN // Check time range
					DiagCode			:= 16#F025;
					Diag.ErrorConfig	:= TRUE;
					Diag.DiagText		:= 'MonitorTimeTooLong';
				END_IF

			//#################### Check the setup of Output Current monitor ##################
			ELSIF ( Config.Current.EnableMon AND NOT(Diag.ErrorConfig) ) THEN
				IF ( ADR(pSO_In_OutputCurrentOK) = 0 ) THEN
					DiagCode			:= 16#F014;
					Diag.ErrorConfig	:= TRUE;
					Diag.DiagText		:= 'NoOutputCurrentOkADR';
				ELSIF ( Config.Current.MonitorTime = 0 ) THEN // Check time range
					DiagCode			:= 16#F024;
					Diag.ErrorConfig	:= TRUE;
					Diag.DiagText		:= 'NoMonitorTime';
				ELSIF ( Config.Current.MonitorTime > T#2s ) THEN // Check time range
					DiagCode			:= 16#F025;
					Diag.ErrorConfig	:= TRUE;
					Diag.DiagText		:= 'MonitorTimeTooLong';
				END_IF

			//#################### Check the setup of Output Interlock monitor ##################
			ELSIF ( Config.InterlockState.EnableMon AND NOT(Diag.ErrorConfig) ) THEN
				IF ( ADR(pSO_In_OutputInterlockStates) = 0 ) THEN
					DiagCode			:= 16#F016;
					Diag.ErrorConfig	:= TRUE;
					Diag.DiagText		:= 'NoOutputInterlockStateADR';
				ELSIF ( Config.InterlockState.MonitorTime = 0 ) THEN // Check time range
					DiagCode			:= 16#F024;
					Diag.ErrorConfig	:= TRUE;
					Diag.DiagText		:= 'NoMonitorTime';
				ELSIF ( Config.InterlockState.MonitorTime > T#1s ) THEN // Check time range
					DiagCode			:= 16#F025;
					Diag.ErrorConfig	:= TRUE;
					Diag.DiagText		:= 'MonitorTimeTooLong';
				ELSIF ( (Config.InterlockState.ChannelSelector < 1) OR (Config.InterlockState.ChannelSelector > 4)) THEN
					DiagCode			:= 16#F026;
					Diag.ErrorConfig	:= TRUE;
					Diag.DiagText		:= 'InvalidOutputInterlockChannelSelector';
				END_IF
			END_IF

			//#################### SUCCESS!!! ##################
			IF NOT( Diag.ErrorConfig ) THEN
				Internal.StateGoTo	:= SC_INIT;
			END_IF

		SC_INIT:
			StateAction_Init;

		SC_DISABLED:
			StateAction_Disabled;

		SC_ENABLED:
			StateAction_Enabled;

		SC_ERROR:
			StateAction_Error;

		ELSE
			//The code should not end uzp here. Report the error as unknown.
			Diag.ErrorInternal	:= TRUE;
			DiagCode			:= 16#CFFF;
			Diag.DiagText		:= 'UndocumentedError';

	END_CASE

	//########## Update fub outputs ##########
	// Update fub error output
	Error := Diag.ErrorSafeFub OR Diag.ErrorInterlock OR Diag.ErrorCurrent OR Diag.ErrorFdbk OR Diag.ErrorConfig OR Diag.ErrorInternal;

	// Update fub IO status outputs
	IF ( Internal.State > SC_INIT ) THEN
		// Update IOSP outputs after fub init is successful, so all safety outputs are in a safe state before energizing and monitoring
		Internal.Output.SO_Out_Contactor1	:= Cmd.OutputRequest;
		Internal.Output.SO_Out_Contactor2	:= Cmd.OutputRequest;

		// Update fub status outputs based on IOSP dual-channel agreement
		Status.OutputActive		:= Internal.Input.SO_In_Output1PhysicalState AND Internal.Input.SO_In_Output2PhysicalState; // both channels need to activate to energize, so all dual-channel diagreements are treated as inactive
		Status.OutputRequested	:= Internal.Output.SO_Out_Contactor1 AND Internal.Output.SO_Out_Contactor2; // both channels need to activate to energize, so all dual-channel diagreements are treated as no request
	ELSE
		// disable IOSP output during CFG state or ERROR state
		Internal.Output.SO_Out_Contactor1	:= FALSE;
		Internal.Output.SO_Out_Contactor2	:= FALSE;

		// Update fub status output based on available SDigitalOut single-channel IOSP data
		Status.OutputActive		:= Internal.Input.SO_In_Output1PhysicalState; // Because there is only one channel, SDigitalOut can always show status based on Internal.Input.SO_In_Output1PhysicalState
		Status.OutputRequested	:= FALSE;
	END_IF

	// Disable internal EDM reset request after a jump out of init state that's not made within the state machine (presumably into error state)
	// Note: Error state sets internal EDM reset request on rising edge of error acknowledgement, so error state needs to disable EDM reset on its own
	IF ( Internal.Prev.State = SC_INIT AND Internal.State <> SC_INIT ) THEN
		Internal.EDMReset	:= FALSE;
	END_IF
	// Pass through safety reset request in all fub states
	Status.SafetyResetRequested	:= Cmd.Reset OR Internal.EDMReset;

	//########## SDigitalOut single-channel simulation output handling ##########
	IF ( Cmd.Simulation.EnableSim ) THEN
		//########## Output destination assignment ##########
		Simulation.Output.SO_Out_Contactor1	:= Internal.Output.SO_Out_Contactor1;
		Simulation.Output.SO_Out_Contactor2	:= Internal.Output.SO_Out_Contactor2;
		//########## Reset real outputs ##########
		IF ( ADR(pSO_Out_DigitalOut) > 0 ) THEN
			pSO_Out_DigitalOut	:= FALSE;
		END_IF
	ELSE
		//########## Output destination assignment ##########
		IF ( ADR(pSO_Out_DigitalOut) > 0 ) THEN
			pSO_Out_DigitalOut	:= Internal.Output.SO_Out_Contactor1;
		END_IF
		//########## Reset simulation outputs ##########
		Simulation.Output.SO_Out_Contactor1	:= FALSE;
		Simulation.Output.SO_Out_Contactor2	:= FALSE;
	END_IF

	//########## Update internal process ##########
	StateAction_CommmonAft;

END_FUNCTION_BLOCK

(* ---- SfContactor.st ---- *)
(*
This fub has four monitoring options, ordered by priority below:
1) SF_EDM DiagCode from safety CPU (highest priority)
2) external contactor state monitoring (using SafeDigitalInput0x from SI card)
3) internal contactor wiring monitoring (using CurrentOK0x from SO card)
4) output interlock state monitoring (using FBOutputState0x0y from SO card) (lowest priority)
If more than one monitoring options are enabled, the highest priority option will be used by the fub to evaluate contactor open/close behavior.
##################################################*)

FUNCTION_BLOCK SfContactor

	//########## Simulation input handling ##########
	IF ( Cmd.Simulation.EnableSim ) THEN
		Simulation.Input.SI_In_SafeModuleOK	:= TRUE;
		Simulation.Input.SO_In_SafeModuleOK	:= TRUE;

		Internal.i	:= TIME_TO_UDINT( clock_ms() ) MOD 200;

		//########## SContactor dual-channel input simulation ##########
		// SimMonitorErrors bits (when set to TRUE):
		//  0: output 1 blocked by safety (interlock)
		//  1: output 2 blocked by safety (interlock)
		//  2: output 1 wire break (current)
		//  3: output 2 wire break (current)
		//  4: fdbk 1 stuck on high/"contactor open" (fdbk)
		//  5: fdbk 2 stuck on high/"contactor open" (fdbk)
		//  6: fdbk 1 stuck on low/"contactor closed" (fdbk)
		//  7: fdbk 2 stuck on low/"contactor closed" (fdbk)

		// simulate interlock feedback
		IF ( Cmd.Simulation.SimMonitorErrors.0 ) THEN
			Simulation.Input.SO_In_Output1PhysicalState	:= FALSE;
			Simulation.Input.InterlockStateOutput1		:= 8;
		ELSE
			Simulation.Input.SO_In_Output1PhysicalState	:= Simulation.Output.SO_Out_Contactor1 AND ( Simulation.Input.SO_In_Output1PhysicalState OR ( Internal.i >= 0	AND Internal.i < 50 ) );
			IF ( Simulation.Input.SO_In_Output1PhysicalState ) THEN
				Simulation.Input.InterlockStateOutput1	:= 9;
			ELSE
				Simulation.Input.InterlockStateOutput1	:= 7;
			END_IF
		END_IF
		IF ( Cmd.Simulation.SimMonitorErrors.1 ) THEN
			Simulation.Input.SO_In_Output2PhysicalState	:= FALSE;
			Simulation.Input.InterlockStateOutput2		:= 8;
		ELSE
			Simulation.Input.SO_In_Output2PhysicalState	:= Simulation.Output.SO_Out_Contactor2 AND ( Simulation.Input.SO_In_Output2PhysicalState OR ( Internal.i >= 15	AND Internal.i < 65 ) );
			IF ( Simulation.Input.SO_In_Output2PhysicalState ) THEN
				Simulation.Input.InterlockStateOutput2	:= 9;
			ELSE
				Simulation.Input.InterlockStateOutput2	:= 7;
			END_IF
		END_IF

		// simulate current ok feedback
		IF ( Cmd.Simulation.SimMonitorErrors.2 ) THEN
			Simulation.Input.SO_In_Output1CurrentOK	:= FALSE;
		ELSE
			Simulation.Input.SO_In_Output1CurrentOK	:= Simulation.Input.SO_In_Output1PhysicalState AND ( Simulation.Input.SO_In_Output1CurrentOK OR ( Internal.i >= 30	AND Internal.i < 80 ) );
		END_IF
		IF ( Cmd.Simulation.SimMonitorErrors.3 ) THEN
			Simulation.Input.SO_In_Output2CurrentOK	:= FALSE;
		ELSE
			Simulation.Input.SO_In_Output2CurrentOK	:= Simulation.Input.SO_In_Output2PhysicalState AND ( Simulation.Input.SO_In_Output2CurrentOK OR ( Internal.i >= 45	AND Internal.i < 95 ) );
		END_IF

		// simulate external monitoring feedback
		IF ( Cmd.Simulation.SimMonitorErrors.4 ) THEN
			Simulation.Input.SI_In_Contactor1Fdbk	:= TRUE;
		ELSIF ( Cmd.Simulation.SimMonitorErrors.6 ) THEN
			Simulation.Input.SI_In_Contactor1Fdbk	:= FALSE;
		ELSE
			IF ( Internal.i >= 60 AND Internal.i < 110 ) THEN
				IF ( Simulation.Input.SO_In_Output1CurrentOK ) THEN
					Simulation.Input.SI_In_Contactor1Fdbk	:= FALSE;
				ELSE
					Simulation.Input.SI_In_Contactor1Fdbk	:= TRUE;
				END_IF
			END_IF
		END_IF
		IF ( Cmd.Simulation.SimMonitorErrors.5 ) THEN
			Simulation.Input.SI_In_Contactor2Fdbk	:= TRUE;
		ELSIF ( Cmd.Simulation.SimMonitorErrors.7 ) THEN
			Simulation.Input.SI_In_Contactor2Fdbk	:= FALSE;
		ELSE
			IF ( Internal.i >= 75 AND Internal.i < 125 ) THEN
				IF ( Simulation.Input.SO_In_Output2CurrentOK ) THEN
					Simulation.Input.SI_In_Contactor2Fdbk	:= FALSE;
				ELSE
					Simulation.Input.SI_In_Contactor2Fdbk	:= TRUE;
				END_IF
			END_IF
		END_IF

		//########## DiagCode simulation ##########
		SimAction_DiagCode;

		//########## SContactor dual-channel input source assignment ##########
		Internal.Input.SF_In_DiagCode		:= Simulation.Input.SF_In_DiagCode;
		Internal.Input.SI_In_SafeModuleOK		:= Simulation.Input.SI_In_SafeModuleOK;
		Internal.Input.SI_In_Contactor1Fdbk		:= Simulation.Input.SI_In_Contactor1Fdbk;
		Internal.Input.SI_In_Contactor2Fdbk		:= Simulation.Input.SI_In_Contactor2Fdbk;
		Internal.Input.SO_In_SafeModuleOK			:= Simulation.Input.SO_In_SafeModuleOK;
		Internal.Input.SO_In_Output1PhysicalState	:= Simulation.Input.SO_In_Output1PhysicalState;
		Internal.Input.SO_In_Output2PhysicalState	:= Simulation.Input.SO_In_Output2PhysicalState;
		Internal.Input.SO_In_Output1CurrentOK		:= Simulation.Input.SO_In_Output1CurrentOK;
		Internal.Input.SO_In_Output2CurrentOK		:= Simulation.Input.SO_In_Output2CurrentOK;
		Internal.Input.SO_In_OutputInterlockStates	:= Simulation.Input.InterlockStateOutput1 + Simulation.Input.InterlockStateOutput2 * 16#10;

	ELSE
		//########## SContactor dual-channel input source assignment ##########
		IF ( ADR(pSF_In_DiagCode) > 0 ) THEN
			Internal.Input.SF_In_DiagCode		:= pSF_In_DiagCode;
		ELSE
			Internal.Input.SF_In_DiagCode		:= 0;
		END_IF
		IF ( ADR(pSI_In_SafeModuleOK) > 0 ) THEN
			Internal.Input.SI_In_SafeModuleOK	:= pSI_In_SafeModuleOK;
		ELSE
			Internal.Input.SI_In_SafeModuleOK	:= 0;
		END_IF
		IF ( ADR(pSI_In_Contactor1Fdbk) > 0 ) THEN
			Internal.Input.SI_In_Contactor1Fdbk	:= pSI_In_Contactor1Fdbk;
		ELSE
			Internal.Input.SI_In_Contactor1Fdbk	:= 0;
		END_IF
		IF ( ADR(pSI_In_Contactor2Fdbk) > 0 ) THEN
			Internal.Input.SI_In_Contactor2Fdbk	:= pSI_In_Contactor2Fdbk;
		ELSE
			Internal.Input.SI_In_Contactor2Fdbk	:= 0;
		END_IF
		IF ( ADR(pSO_In_SafeModuleOK) > 0 ) THEN
			Internal.Input.SO_In_SafeModuleOK			:= pSO_In_SafeModuleOK;
		ELSE
			Internal.Input.SO_In_SafeModuleOK			:= 0;
		END_IF
		IF ( ADR(pSO_In_Output1PhysicalState) > 0 ) THEN
			Internal.Input.SO_In_Output1PhysicalState	:= pSO_In_Output1PhysicalState;
		ELSE
			Internal.Input.SO_In_Output1PhysicalState	:= 0;
		END_IF
		IF ( ADR(pSO_In_Output2PhysicalState) > 0 ) THEN
			Internal.Input.SO_In_Output2PhysicalState	:= pSO_In_Output2PhysicalState;
		ELSE
			Internal.Input.SO_In_Output2PhysicalState	:= 0;
		END_IF
		IF ( ADR(pSO_In_Output1CurrentOK) > 0 ) THEN
			Internal.Input.SO_In_Output1CurrentOK		:= pSO_In_Output1CurrentOK;
		ELSE
			Internal.Input.SO_In_Output1CurrentOK		:= 0;
		END_IF
		IF ( ADR(pSO_In_Output2CurrentOK) > 0 ) THEN
			Internal.Input.SO_In_Output2CurrentOK		:= pSO_In_Output2CurrentOK;
		ELSE
			Internal.Input.SO_In_Output2CurrentOK		:= 0;
		END_IF
		IF ( ADR(pSO_In_OutputInterlockStates) > 0 ) THEN
			Internal.Input.SO_In_OutputInterlockStates	:= pSO_In_OutputInterlockStates;
		ELSE
			Internal.Input.SO_In_OutputInterlockStates	:= 0;
		END_IF
		//########## Reset simulation inputs ##########
		brsmemset( ADR(Simulation.Input), 0, SIZEOF(Simulation.Input) );

	END_IF

	//########## SContactor dual-channel output interlock state identification ##########
	// Read output channel interlock state
	IF ( Config.InterlockState.EnableMon ) THEN
		Internal.Input.InterlockStateOutput1 := Internal.Input.SO_In_OutputInterlockStates AND 16#0F;
		Internal.Input.InterlockStateOutput2 := SHR(( Internal.Input.SO_In_OutputInterlockStates AND 16#F0 ), 4);
	ELSE
		Internal.Input.InterlockStateOutput1 := 0;
		Internal.Input.InterlockStateOutput2 := 0;
	END_IF

	//########## Feedback interpretation and error state transition ##########
	StateAction_CommonPre;

	//########## State machine for processing feedback values ##########
	CASE Internal.State OF

		SC_CFG:
			//#################### Req. Checkout ####################
			IF ( ADR(pSO_In_SafeModuleOK) = 0 ) THEN // Check if the monitoring of safe communication to SO node exists
				DiagCode			:= 16#F001;
				Diag.ErrorConfig	:= TRUE;
				Diag.DiagText		:= 'NoSafeDOCardOkADR';
			ELSIF ( ADR(pSO_Out_Contactor1) = 0 ) THEN // Check if output channe l exists
				DiagCode			:= 16#F002;
				Diag.ErrorConfig	:= TRUE;
				Diag.DiagText		:= 'NoContactor1OutADR';
			ELSIF ( ADR(pSO_Out_Contactor2) = 0 ) THEN // Check if output channe 2 exists
				DiagCode			:= 16#F003;
				Diag.ErrorConfig	:= TRUE;
				Diag.DiagText		:= 'NoContactor2OutADR';
			ELSIF ( ADR(pSO_In_Output1PhysicalState) = 0 ) THEN // Check if the output phsical state monitoring exists
				DiagCode			:= 16#F004;
				Diag.ErrorConfig	:= TRUE;
				Diag.DiagText		:= 'NoOutput1PhysicalStateADR';
			ELSIF ( ADR(pSO_In_Output2PhysicalState) = 0 ) THEN // Check if the output phsical state monitoring exists
				DiagCode			:= 16#F005;
				Diag.ErrorConfig	:= TRUE;
				Diag.DiagText		:= 'NoOutput2PhysicalStateADR';
			END_IF
			// No MonitorTime for PhysicalState because we don't know when the safety CPU will approve output enable request

			//#################### Check the setup of safety-to-gray comm of SF_EDM fub DiagCode monitor ##################
			IF ( Config.DiagCode.EnableMon AND NOT(Diag.ErrorConfig) ) THEN
				IF ( ADR(pSF_In_DiagCode) = 0 ) THEN // Check if the monitoring of DiagCode from safety CPU exists
					DiagCode			:= 16#F010;
					Diag.ErrorConfig	:= TRUE;
					Diag.DiagText		:= 'NoDiagCodeADR';
				ELSIF ( ADR(pSI_In_SafeModuleOK) = 0 ) THEN // Check if the monitoring of safe communication to SI node exists
					DiagCode			:= 16#F011;
					Diag.ErrorConfig	:= TRUE;
					Diag.DiagText		:= 'NoSafeDICardOkADR';
				ELSIF ( ADR(pSI_In_Contactor1Fdbk) = 0 ) THEN // Need an SI card input to monitor
					DiagCode			:= 16#F012;
					Diag.ErrorConfig	:= TRUE;
					Diag.DiagText		:= 'NoContactor1FdbkADR';
				ELSIF ( ADR(pSI_In_Contactor2Fdbk) = 0 ) THEN // Need an SI card input to monitor
					DiagCode			:= 16#F013;
					Diag.ErrorConfig	:= TRUE;
					Diag.DiagText		:= 'NoContactor2FdbkADR';
				ELSIF ( Config.DiagCode.StartDelayTime = 0 ) THEN // Check time range
					DiagCode			:= 16#F020;
					Diag.ErrorConfig	:= TRUE;
					Diag.DiagText		:= 'NoStartDelay';
				ELSIF ( Config.DiagCode.StartDelayTime > T#2m ) THEN // Check time range
					DiagCode			:= 16#F021;
					Diag.ErrorConfig	:= TRUE;
					Diag.DiagText		:= 'StartDelayTooLong';
				ELSIF ( Config.DiagCode.ResetDelayTime = 0 ) THEN // Check time range
					DiagCode			:= 16#F022;
					Diag.ErrorConfig	:= TRUE;
					Diag.DiagText		:= 'NoResetDelay';
				ELSIF ( Config.DiagCode.ResetDelayTime > T#10s ) THEN // Check time range
					DiagCode			:= 16#F023;
					Diag.ErrorConfig	:= TRUE;
					Diag.DiagText		:= 'ResetDelayTooLong';
				END_IF

			//#################### Check the setup of Contactor Feedback monitor ####################
			ELSIF ( Config.Fdbk.EnableMon AND NOT(Diag.ErrorConfig) ) THEN
				IF ( ADR(pSI_In_SafeModuleOK) = 0 ) THEN // Check if the monitoring of safe communication to SI node exists
					DiagCode			:= 16#F011;
					Diag.ErrorConfig	:= TRUE;
					Diag.DiagText		:= 'NoSafeDICardOkADR';
				ELSIF ( ADR(pSI_In_Contactor1Fdbk) = 0 ) THEN // Need an SI card input to monitor
					DiagCode			:= 16#F012;
					Diag.ErrorConfig	:= TRUE;
					Diag.DiagText		:= 'NoContactor1FdbkADR';
				ELSIF ( ADR(pSI_In_Contactor2Fdbk) = 0 ) THEN // Need an SI card input to monitor
					DiagCode			:= 16#F013;
					Diag.ErrorConfig	:= TRUE;
					Diag.DiagText		:= 'NoContactor2FdbkADR';
				ELSIF ( Config.Fdbk.StartDelayTime = 0 ) THEN // Check time range
					DiagCode			:= 16#F020;
					Diag.ErrorConfig	:= TRUE;
					Diag.DiagText		:= 'NoStartDelay';
				ELSIF ( Config.Fdbk.StartDelayTime > T#10s ) THEN // Check time range
					DiagCode			:= 16#F021;
					Diag.ErrorConfig	:= TRUE;
					Diag.DiagText		:= 'StartDelayTooLong';
				ELSIF ( Config.Fdbk.MonitorTime = 0 ) THEN // Check time range
					DiagCode			:= 16#F024;
					Diag.ErrorConfig	:= TRUE;
					Diag.DiagText		:= 'NoMonitorTime';
				ELSIF ( Config.Fdbk.MonitorTime > T#2s ) THEN // Check time range
					DiagCode			:= 16#F025;
					Diag.ErrorConfig	:= TRUE;
					Diag.DiagText		:= 'MonitorTimeTooLong';
				END_IF

			//#################### Check the setup of Output Current monitor ##################
			ELSIF ( Config.Current.EnableMon AND NOT(Diag.ErrorConfig) ) THEN
				IF ( ADR(pSO_In_Output1CurrentOK) = 0 ) THEN
					DiagCode			:= 16#F014;
					Diag.ErrorConfig	:= TRUE;
					Diag.DiagText		:= 'NoOutput1CurrentOkADR';
				ELSIF ( ADR(pSO_In_Output2CurrentOK) = 0 ) THEN
					DiagCode			:= 16#F015;
					Diag.ErrorConfig	:= TRUE;
					Diag.DiagText		:= 'NoOutput2CurrentOkADR';
				ELSIF ( Config.Current.MonitorTime = 0 ) THEN // Check time range
					DiagCode			:= 16#F024;
					Diag.ErrorConfig	:= TRUE;
					Diag.DiagText		:= 'NoMonitorTime';
				ELSIF ( Config.Current.MonitorTime > T#2s ) THEN // Check time range
					DiagCode			:= 16#F025;
					Diag.ErrorConfig	:= TRUE;
					Diag.DiagText		:= 'MonitorTimeTooLong';
				END_IF

			//#################### Check the setup of Output Interlock monitor ##################
			ELSIF ( Config.InterlockState.EnableMon AND NOT(Diag.ErrorConfig) ) THEN
				IF ( ADR(pSO_In_OutputInterlockStates) = 0 ) THEN
					DiagCode			:= 16#F016;
					Diag.ErrorConfig	:= TRUE;
					Diag.DiagText		:= 'NoOutputInterlockStateADR';
				ELSIF ( Config.InterlockState.MonitorTime = 0 ) THEN // Check time range
					DiagCode			:= 16#F024;
					Diag.ErrorConfig	:= TRUE;
					Diag.DiagText		:= 'NoMonitorTime';
				ELSIF ( Config.InterlockState.MonitorTime > T#1s ) THEN // Check time range
					DiagCode			:= 16#F025;
					Diag.ErrorConfig	:= TRUE;
					Diag.DiagText		:= 'MonitorTimeTooLong';
				END_IF
			END_IF

			//#################### SUCCESS!!! ##################
			IF NOT( Diag.ErrorConfig ) THEN
				Internal.StateGoTo	:= SC_INIT;
			END_IF

		SC_INIT:
			StateAction_Init;

		SC_DISABLED:
			StateAction_Disabled;

		SC_ENABLED:
			StateAction_Enabled;

		SC_ERROR:
			StateAction_Error;

		ELSE
			//The code should not end uzp here. Report the error as unknown.
			Diag.ErrorInternal	:= TRUE;
			DiagCode			:= 16#CFFF;
			Diag.DiagText		:= 'UndocumentedError';

	END_CASE

	//########## Update fub outputs ##########
	// Update fub error output
	Error := Diag.ErrorSafeFub OR Diag.ErrorInterlock OR Diag.ErrorCurrent OR Diag.ErrorFdbk OR Diag.ErrorConfig OR Diag.ErrorInternal;

	// Update fub IO status outputs
	IF ( Internal.State > SC_INIT ) THEN
		// Update IOSP outputs after fub init is successful, so all safety outputs are in a safe state before energizing and monitoring
		Internal.Output.SO_Out_Contactor1	:= Cmd.OutputRequest;
		Internal.Output.SO_Out_Contactor2	:= Cmd.OutputRequest;

		// Update fub status outputs based on IOSP dual-channel agreement
		Status.OutputActive		:= Internal.Input.SO_In_Output1PhysicalState AND Internal.Input.SO_In_Output2PhysicalState; // both channels need to activate to energize, so all dual-channel diagreements are treated as inactive
		Status.OutputRequested	:= Internal.Output.SO_Out_Contactor1 AND Internal.Output.SO_Out_Contactor2; // both channels need to activate to energize, so all dual-channel diagreements are treated as no request
	ELSE
		// disable IOSP output during CFG state or ERROR state
		Internal.Output.SO_Out_Contactor1	:= FALSE;
		Internal.Output.SO_Out_Contactor2	:= FALSE;

		// Update fub status output based on available SContactor dual-channel IOSP data
		IF ( ADR(pSO_In_Output1PhysicalState) > 0 AND ADR(pSO_In_Output2PhysicalState) > 0 ) THEN
			Status.OutputActive	:= Internal.Input.SO_In_Output1PhysicalState AND Internal.Input.SO_In_Output2PhysicalState;
		ELSIF ( ADR(pSO_In_Output1PhysicalState) > 0 ) THEN
			Status.OutputActive	:= Internal.Input.SO_In_Output1PhysicalState;
		ELSIF ( ADR(pSO_In_Output2PhysicalState) > 0 ) THEN
			Status.OutputActive	:= Internal.Input.SO_In_Output2PhysicalState;
		ELSE
			Status.OutputActive	:= FALSE;
		END_IF
		Status.OutputRequested	:= FALSE;
	END_IF

	// Disable internal EDM reset request after a jump out of init state that's not made within the state machine (presumably into error state)
	// Note: Error state sets internal EDM reset request on rising edge of error acknowledgement, so error state needs to disable EDM reset on its own
	IF ( Internal.Prev.State = SC_INIT AND Internal.State <> SC_INIT ) THEN
		Internal.EDMReset	:= FALSE;
	END_IF
	// Pass through safety reset request in all fub states
	Status.SafetyResetRequested	:= Cmd.Reset OR Internal.EDMReset;

	//########## SContactor dual-channel Simulation output handling ##########
	IF ( Cmd.Simulation.EnableSim ) THEN
		//########## Output destination assignment ##########
		Simulation.Output.SO_Out_Contactor1	:= Internal.Output.SO_Out_Contactor1;
		Simulation.Output.SO_Out_Contactor2	:= Internal.Output.SO_Out_Contactor2;
		//########## Reset real outputs ##########
		IF ( ADR(pSO_Out_Contactor1) > 0 ) THEN
			pSO_Out_Contactor1	:= FALSE;
		END_IF
		IF ( ADR(pSO_Out_Contactor2) > 0 ) THEN
			pSO_Out_Contactor2	:= FALSE;
		END_IF
	ELSE
		//########## Output destination assignment ##########
		IF ( ADR(pSO_Out_Contactor1) > 0 ) THEN
			pSO_Out_Contactor1	:= Internal.Output.SO_Out_Contactor1;
		END_IF
		IF ( ADR(pSO_Out_Contactor2) > 0 ) THEN
			pSO_Out_Contactor2	:= Internal.Output.SO_Out_Contactor2;
		END_IF
		//########## Reset simulation outputs ##########
		Simulation.Output.SO_Out_Contactor1	:= FALSE;
		Simulation.Output.SO_Out_Contactor2	:= FALSE;
	END_IF

	//########## Update internal process ##########
	StateAction_CommmonAft;

END_FUNCTION_BLOCK

(* ---- SfDigitalOut.st ---- *)
(*
This fub has four monitoring options, ordered by priority below:
1) SF_EDM DiagCode from safety CPU (highest priority)
2) external contactor state monitoring (using SafeDigitalInput0x from SI card)
3) internal contactor wiring monitoring (using CurrentOK0x from SO card)
4) output interlock state monitoring (using FBOutputState0x0y from SO card) (lowest priority)
If more than one monitoring options are enabled, the highest priority option will be used by the fub to evaluate contactor open/close behavior.
##################################################*)

FUNCTION_BLOCK SfDigitalOut

	//########## Simulation input handling ##########
	IF ( Cmd.Simulation.EnableSim ) THEN
		Simulation.Input.SI_In_SafeModuleOK	:= TRUE;
		Simulation.Input.SO_In_SafeModuleOK	:= TRUE;

		Internal.i	:= TIME_TO_UDINT( clock_ms() ) MOD 200;

		//########## SDigitalOut single-channel input simulation ##########
		// SimMonitorErrors bits (when set to TRUE):
		//  0: output X blocked by safety (interlock)
		//  1: output X blocked by safety (interlock)
		//  2: output X wire break (current)
		//  3: output X wire break (current)
		//  4: fdbk X stuck on high/"contactor open" (fdbk)
		//  5: fdbk X stuck on high/"contactor open" (fdbk)
		//  6: fdbk X stuck on low/"contactor closed" (fdbk)
		//  7: fdbk X stuck on low/"contactor closed" (fdbk)

		// simulate interlock feedback
		IF ( Cmd.Simulation.SimMonitorErrors.0 OR Cmd.Simulation.SimMonitorErrors.1 ) THEN
			Simulation.Input.SO_In_Output1PhysicalState	:= FALSE;
			Simulation.Input.InterlockStateOutput1		:= 8;
		ELSE
			Simulation.Input.SO_In_Output1PhysicalState	:= Simulation.Output.SO_Out_Contactor1 AND ( Simulation.Input.SO_In_Output1PhysicalState OR ( Internal.i >= 0	AND Internal.i < 50 ) );
			IF ( Simulation.Input.SO_In_Output1PhysicalState ) THEN
				Simulation.Input.InterlockStateOutput1	:= 9;
			ELSE
				Simulation.Input.InterlockStateOutput1	:= 7;
			END_IF
		END_IF

		// simulate current ok feedback
		IF ( Cmd.Simulation.SimMonitorErrors.2 OR Cmd.Simulation.SimMonitorErrors.3 ) THEN
			Simulation.Input.SO_In_Output1CurrentOK	:= FALSE;
		ELSE
			Simulation.Input.SO_In_Output1CurrentOK	:= Simulation.Input.SO_In_Output1PhysicalState AND ( Simulation.Input.SO_In_Output1CurrentOK OR ( Internal.i >= 30	AND Internal.i < 80 ) );
		END_IF

		// simulate external monitoring feedback
		IF ( Cmd.Simulation.SimMonitorErrors.4 OR Cmd.Simulation.SimMonitorErrors.5 ) THEN
			Simulation.Input.SI_In_Contactor1Fdbk	:= TRUE;
		ELSIF ( Cmd.Simulation.SimMonitorErrors.6 OR Cmd.Simulation.SimMonitorErrors.7 ) THEN
			Simulation.Input.SI_In_Contactor1Fdbk	:= FALSE;
		ELSE
			IF ( Internal.i >= 60 AND Internal.i < 110 ) THEN
				IF ( Simulation.Input.SO_In_Output1CurrentOK ) THEN
					Simulation.Input.SI_In_Contactor1Fdbk	:= FALSE;
				ELSE
					Simulation.Input.SI_In_Contactor1Fdbk	:= TRUE;
				END_IF
			END_IF
		END_IF
		Simulation.Input.SI_In_Contactor2Fdbk		:= Simulation.Input.SI_In_Contactor1Fdbk;
		Simulation.Input.SO_In_Output2PhysicalState	:= Simulation.Input.SO_In_Output1PhysicalState;
		Simulation.Input.SO_In_Output2CurrentOK		:= Simulation.Input.SO_In_Output1CurrentOK;
		Simulation.Input.InterlockStateOutput2		:= Simulation.Input.InterlockStateOutput1;

		//########## DiagCode simulation ##########
		SimAction_DiagCode;

		//########## SDigitalOut single-channel input source assignment ##########
		Internal.Input.SF_In_DiagCode		:= Simulation.Input.SF_In_DiagCode;
		Internal.Input.SI_In_SafeModuleOK		:= Simulation.Input.SI_In_SafeModuleOK;
		Internal.Input.SI_In_Contactor1Fdbk		:= Simulation.Input.SI_In_Contactor1Fdbk;
		Internal.Input.SI_In_Contactor2Fdbk		:= Simulation.Input.SI_In_Contactor2Fdbk;
		Internal.Input.SO_In_SafeModuleOK			:= Simulation.Input.SO_In_SafeModuleOK;
		Internal.Input.SO_In_Output1PhysicalState	:= Simulation.Input.SO_In_Output1PhysicalState;
		Internal.Input.SO_In_Output2PhysicalState	:= Simulation.Input.SO_In_Output2PhysicalState;
		Internal.Input.SO_In_Output1CurrentOK		:= Simulation.Input.SO_In_Output1CurrentOK;
		Internal.Input.SO_In_Output2CurrentOK		:= Simulation.Input.SO_In_Output2CurrentOK;
		CASE Config.InterlockState.ChannelSelector OF
			1:
				Internal.Input.SO_In_OutputInterlockStates	:= Simulation.Input.InterlockStateOutput1;
			2:
				Internal.Input.SO_In_OutputInterlockStates	:= Simulation.Input.InterlockStateOutput1 * 16#10;
			ELSE
				Internal.Input.SO_In_OutputInterlockStates	:= 0;
		END_CASE

	ELSE
		//########## SDigitalOut single-channel input source assignment ##########
		IF ( ADR(pSF_In_DiagCode) > 0 ) THEN
			Internal.Input.SF_In_DiagCode		:= pSF_In_DiagCode;
		ELSE
			Internal.Input.SF_In_DiagCode		:= 0;
		END_IF
		IF ( ADR(pSI_In_SafeModuleOK) > 0 ) THEN
			Internal.Input.SI_In_SafeModuleOK	:= pSI_In_SafeModuleOK;
		ELSE
			Internal.Input.SI_In_SafeModuleOK	:= 0;
		END_IF
		IF ( ADR(pSI_In_DigitalOutFdbk) > 0 ) THEN
			Internal.Input.SI_In_Contactor1Fdbk	:= pSI_In_DigitalOutFdbk;
		ELSE
			Internal.Input.SI_In_Contactor1Fdbk	:= 0;
		END_IF
		IF ( ADR(pSO_In_SafeModuleOK) > 0 ) THEN
			Internal.Input.SO_In_SafeModuleOK			:= pSO_In_SafeModuleOK;
		ELSE
			Internal.Input.SO_In_SafeModuleOK			:= 0;
		END_IF
		IF ( ADR(pSO_In_OutputPhysicalState) > 0 ) THEN
			Internal.Input.SO_In_Output1PhysicalState	:= pSO_In_OutputPhysicalState;
		ELSE
			Internal.Input.SO_In_Output1PhysicalState	:= 0;
		END_IF
		IF ( ADR(pSO_In_OutputCurrentOK) > 0 ) THEN
			Internal.Input.SO_In_Output1CurrentOK		:= pSO_In_OutputCurrentOK;
		ELSE
			Internal.Input.SO_In_Output1CurrentOK		:= 0;
		END_IF
		IF ( ADR(pSO_In_OutputInterlockStates) > 0 ) THEN
			Internal.Input.SO_In_OutputInterlockStates	:= pSO_In_OutputInterlockStates;
		ELSE
			Internal.Input.SO_In_OutputInterlockStates	:= 0;
		END_IF
		Internal.Input.SI_In_Contactor2Fdbk			:= Internal.Input.SI_In_Contactor1Fdbk;
		Internal.Input.SO_In_Output2PhysicalState	:= Internal.Input.SO_In_Output1PhysicalState;
		Internal.Input.SO_In_Output2CurrentOK		:= Internal.Input.SO_In_Output1CurrentOK;
		//########## Reset simulation inputs ##########
		brsmemset( ADR(Simulation.Input), 0, SIZEOF(Simulation.Input) );

	END_IF

	//########## SDigitalOut single-channel output interlock state identification ##########
	// Read output channel interlock state
	IF ( Config.InterlockState.EnableMon ) THEN
		CASE Config.InterlockState.ChannelSelector OF
			1:
				Internal.Input.InterlockStateOutput1 := Internal.Input.SO_In_OutputInterlockStates AND 16#0F;
			2:
				Internal.Input.InterlockStateOutput1 := SHR(( Internal.Input.SO_In_OutputInterlockStates AND 16#F0 ), 4);
			ELSE
				Internal.Input.InterlockStateOutput1 := 0;
		END_CASE
	ELSE
		Internal.Input.InterlockStateOutput1 := 0;
	END_IF
	Internal.Input.InterlockStateOutput2 := Internal.Input.InterlockStateOutput1;

	//########## Feedback interpretation and error state transition ##########
	StateAction_CommonPre;

	//########## State machine for processing feedback values ##########
	CASE Internal.State OF

		SC_CFG:
			//#################### Req. Checkout ####################
			IF ( ADR(pSO_In_SafeModuleOK) = 0 ) THEN // Check if the monitoring of safe communication to SO node exists
				DiagCode			:= 16#F001;
				Diag.ErrorConfig	:= TRUE;
				Diag.DiagText		:= 'NoSafeDOCardOkADR';
			ELSIF ( ADR(pSO_Out_DigitalOut) = 0 ) THEN // Check if output channel exists
				DiagCode			:= 16#F002;
				Diag.ErrorConfig	:= TRUE;
				Diag.DiagText		:= 'NoSafeDigitalOutADR';
			ELSIF ( ADR(pSO_In_OutputPhysicalState) = 0 ) THEN // Check if the output phsical state monitoring exists
				DiagCode			:= 16#F004;
				Diag.ErrorConfig	:= TRUE;
				Diag.DiagText		:= 'NoOutputPhysicalStateADR';
			END_IF
			// No MonitorTime for PhysicalState because we don't know when the safety CPU will approve output enable request

			//#################### Check the setup of safety-to-gray comm of SF_EDM fub DiagCode monitor ##################
			IF ( Config.DiagCode.EnableMon AND NOT(Diag.ErrorConfig) ) THEN
				IF ( ADR(pSF_In_DiagCode) = 0 ) THEN // Check if the monitoring of DiagCode from safety CPU exists
					DiagCode			:= 16#F010;
					Diag.ErrorConfig	:= TRUE;
					Diag.DiagText		:= 'NoDiagCodeADR';
				ELSIF ( ADR(pSI_In_SafeModuleOK) = 0 ) THEN // Check if the monitoring of safe communication to SI node exists
					DiagCode			:= 16#F011;
					Diag.ErrorConfig	:= TRUE;
					Diag.DiagText		:= 'NoSafeDICardOkADR';
				ELSIF ( ADR(pSI_In_DigitalOutFdbk) = 0 ) THEN // Need an SI card input to monitor
					DiagCode			:= 16#F012;
					Diag.ErrorConfig	:= TRUE;
					Diag.DiagText		:= 'NoDigitalOutFdbkADR';
				ELSIF ( Config.DiagCode.StartDelayTime = 0 ) THEN // Check time range
					DiagCode			:= 16#F020;
					Diag.ErrorConfig	:= TRUE;
					Diag.DiagText		:= 'NoStartDelay';
				ELSIF ( Config.DiagCode.StartDelayTime > T#10s ) THEN // Check time range
					DiagCode			:= 16#F021;
					Diag.ErrorConfig	:= TRUE;
					Diag.DiagText		:= 'StartDelayTooLong';
				ELSIF ( Config.DiagCode.ResetDelayTime = 0 ) THEN // Check time range
					DiagCode			:= 16#F022;
					Diag.ErrorConfig	:= TRUE;
					Diag.DiagText		:= 'NoResetDelay';
				ELSIF ( Config.DiagCode.ResetDelayTime > T#10s ) THEN // Check time range
					DiagCode			:= 16#F023;
					Diag.ErrorConfig	:= TRUE;
					Diag.DiagText		:= 'ResetDelayTooLong';
				END_IF

			//#################### Check the setup of Contactor Feedback monitor ####################
			ELSIF ( Config.Fdbk.EnableMon AND NOT(Diag.ErrorConfig) ) THEN
				IF ( ADR(pSI_In_SafeModuleOK) = 0 ) THEN // Check if the monitoring of safe communication to SI node exists
					DiagCode			:= 16#F011;
					Diag.ErrorConfig	:= TRUE;
					Diag.DiagText		:= 'NoSafeDICardOkADR';
				ELSIF ( ADR(pSI_In_DigitalOutFdbk) = 0 ) THEN // Need an SI card input to monitor
					DiagCode			:= 16#F012;
					Diag.ErrorConfig	:= TRUE;
					Diag.DiagText		:= 'NoDigitalOutFdbkADR';
				ELSIF ( Config.Fdbk.StartDelayTime = 0 ) THEN // Check time range
					DiagCode			:= 16#F020;
					Diag.ErrorConfig	:= TRUE;
					Diag.DiagText		:= 'NoStartDelay';
				ELSIF ( Config.Fdbk.StartDelayTime > T#10s ) THEN // Check time range
					DiagCode			:= 16#F021;
					Diag.ErrorConfig	:= TRUE;
					Diag.DiagText		:= 'StartDelayTooLong';
				ELSIF ( Config.Fdbk.MonitorTime = 0 ) THEN // Check time range
					DiagCode			:= 16#F024;
					Diag.ErrorConfig	:= TRUE;
					Diag.DiagText		:= 'NoMonitorTime';
				ELSIF ( Config.Fdbk.MonitorTime > T#2s ) THEN // Check time range
					DiagCode			:= 16#F025;
					Diag.ErrorConfig	:= TRUE;
					Diag.DiagText		:= 'MonitorTimeTooLong';
				END_IF

			//#################### Check the setup of Output Current monitor ##################
			ELSIF ( Config.Current.EnableMon AND NOT(Diag.ErrorConfig) ) THEN
				IF ( ADR(pSO_In_OutputCurrentOK) = 0 ) THEN
					DiagCode			:= 16#F014;
					Diag.ErrorConfig	:= TRUE;
					Diag.DiagText		:= 'NoOutputCurrentOkADR';
				ELSIF ( Config.Current.MonitorTime = 0 ) THEN // Check time range
					DiagCode			:= 16#F024;
					Diag.ErrorConfig	:= TRUE;
					Diag.DiagText		:= 'NoMonitorTime';
				ELSIF ( Config.Current.MonitorTime > T#2s ) THEN // Check time range
					DiagCode			:= 16#F025;
					Diag.ErrorConfig	:= TRUE;
					Diag.DiagText		:= 'MonitorTimeTooLong';
				END_IF

			//#################### Check the setup of Output Interlock monitor ##################
			ELSIF ( Config.InterlockState.EnableMon AND NOT(Diag.ErrorConfig) ) THEN
				IF ( ADR(pSO_In_OutputInterlockStates) = 0 ) THEN
					DiagCode			:= 16#F016;
					Diag.ErrorConfig	:= TRUE;
					Diag.DiagText		:= 'NoOutputInterlockStateADR';
				ELSIF ( Config.InterlockState.MonitorTime = 0 ) THEN // Check time range
					DiagCode			:= 16#F024;
					Diag.ErrorConfig	:= TRUE;
					Diag.DiagText		:= 'NoMonitorTime';
				ELSIF ( Config.InterlockState.MonitorTime > T#1s ) THEN // Check time range
					DiagCode			:= 16#F025;
					Diag.ErrorConfig	:= TRUE;
					Diag.DiagText		:= 'MonitorTimeTooLong';
				ELSIF ( (Config.InterlockState.ChannelSelector < 1) OR (Config.InterlockState.ChannelSelector > 2)) THEN
					DiagCode			:= 16#F026;
					Diag.ErrorConfig	:= TRUE;
					Diag.DiagText		:= 'InvalidOutputInterlockChannelSelector';
				END_IF
			END_IF

			//#################### SUCCESS!!! ##################
			IF NOT( Diag.ErrorConfig ) THEN
				Internal.StateGoTo	:= SC_INIT;
			END_IF

		SC_INIT:
			StateAction_Init;

		SC_DISABLED:
			StateAction_Disabled;

		SC_ENABLED:
			StateAction_Enabled;

		SC_ERROR:
			StateAction_Error;

		ELSE
			//The code should not end uzp here. Report the error as unknown.
			Diag.ErrorInternal	:= TRUE;
			DiagCode			:= 16#CFFF;
			Diag.DiagText		:= 'UndocumentedError';

	END_CASE

	//########## Update fub outputs ##########
	// Update fub error output
	Error := Diag.ErrorSafeFub OR Diag.ErrorInterlock OR Diag.ErrorCurrent OR Diag.ErrorFdbk OR Diag.ErrorConfig OR Diag.ErrorInternal;

	// Update fub IO status outputs
	IF ( Internal.State > SC_INIT ) THEN
		// Update IOSP outputs after fub init is successful, so all safety outputs are in a safe state before energizing and monitoring
		Internal.Output.SO_Out_Contactor1	:= Cmd.OutputRequest;
		Internal.Output.SO_Out_Contactor2	:= Cmd.OutputRequest;

		// Update fub status outputs based on IOSP dual-channel agreement
		Status.OutputActive		:= Internal.Input.SO_In_Output1PhysicalState AND Internal.Input.SO_In_Output2PhysicalState; // both channels need to activate to energize, so all dual-channel diagreements are treated as inactive
		Status.OutputRequested	:= Internal.Output.SO_Out_Contactor1 AND Internal.Output.SO_Out_Contactor2; // both channels need to activate to energize, so all dual-channel diagreements are treated as no request
	ELSE
		// disable IOSP output during CFG state or ERROR state
		Internal.Output.SO_Out_Contactor1	:= FALSE;
		Internal.Output.SO_Out_Contactor2	:= FALSE;

		// Update fub status output based on available SDigitalOut single-channel IOSP data
		Status.OutputActive		:= Internal.Input.SO_In_Output1PhysicalState; // Because there is only one channel, SDigitalOut can always show status based on Internal.Input.SO_In_Output1PhysicalState
		Status.OutputRequested	:= FALSE;
	END_IF

	// Disable internal EDM reset request after a jump out of init state that's not made within the state machine (presumably into error state)
	// Note: Error state sets internal EDM reset request on rising edge of error acknowledgement, so error state needs to disable EDM reset on its own
	IF ( Internal.Prev.State = SC_INIT AND Internal.State <> SC_INIT ) THEN
		Internal.EDMReset	:= FALSE;
	END_IF
	// Pass through safety reset request in all fub states
	Status.SafetyResetRequested	:= Cmd.Reset OR Internal.EDMReset;

	//########## SDigitalOut single-channel simulation output handling ##########
	IF ( Cmd.Simulation.EnableSim ) THEN
		//########## Output destination assignment ##########
		Simulation.Output.SO_Out_Contactor1	:= Internal.Output.SO_Out_Contactor1;
		Simulation.Output.SO_Out_Contactor2	:= Internal.Output.SO_Out_Contactor2;
		//########## Reset real outputs ##########
		IF ( ADR(pSO_Out_DigitalOut) > 0 ) THEN
			pSO_Out_DigitalOut	:= FALSE;
		END_IF
	ELSE
		//########## Output destination assignment ##########
		IF ( ADR(pSO_Out_DigitalOut) > 0 ) THEN
			pSO_Out_DigitalOut	:= Internal.Output.SO_Out_Contactor1;
		END_IF
		//########## Reset simulation outputs ##########
		Simulation.Output.SO_Out_Contactor1	:= FALSE;
		Simulation.Output.SO_Out_Contactor2	:= FALSE;
	END_IF

	//########## Update internal process ##########
	StateAction_CommmonAft;

END_FUNCTION_BLOCK

(* ---- DiagAction_DiagCode.st ---- *)
ACTION DiagAction_DiagCode:

	// Pass through safety CPU's SF_EDM fub DiagCode
	IF ( Internal.Input.SF_In_DiagCode > 0 ) THEN
		// 16#0 is not passed through because whether it is information or error (and require a custom DiagCode display) depends on preexisting fub state and timeout
		DiagCode	:= Internal.Input.SF_In_DiagCode;
	END_IF
	// Go to error state if any error is reported by safety CPU
	IF ( Internal.Input.SF_In_DiagCode >= 16#C000 ) THEN // SF_EDM DiagCode shows an error
		Internal.StateGoTo	:= SC_ERROR;
		Diag.ErrorSafeFub	:= TRUE;
	END_IF

	// Look up custom DiagText
	CASE Internal.Input.SF_In_DiagCode OF
		// 16#0 is not listed because whether it is information or error depends on the fub state and timeout
		// Information
		16#8000:
		Diag.DiagText := 'Energized';
		16#8001:
		Diag.DiagText := 'RequireStartReset';
		16#8010:
		IF NOT( Config.InterlockState.EnableMon ) THEN
			Diag.DiagText := 'RequireOutReq';
		ELSE
			// See Config.InterlockState.EnableMon section
		END_IF
		// Error
		16#C001:
		Diag.DiagText := 'PosReset';
		16#C010:
		Diag.DiagText := 'SameTimePosEdgeOutReqNegEdgeFdbk1';
		16#C011:
		Diag.DiagText := 'SameTimePosEdgeOutReqNegEdgeFdbk1PosReset';
		16#C020:
		Diag.DiagText := 'SameTimePosEdgeOutReqNegEdgeFdbk2';
		16#C021:
		Diag.DiagText := 'SameTimePosEdgeOutReqNegEdgeFdbk2PosReset';
		16#C030:
		Diag.DiagText := 'SameTimePosEdgeOutReqNegEdgeFdbk1Fdbk2';
		16#C031:
		Diag.DiagText := 'SameTimePosEdgeOutReqNegEdgeFdbk1Fdbk2PosReset';
		16#C040:
		Diag.DiagText := 'NegFdbk1AfterNegOutReq';
		16#C041:
		Diag.DiagText := 'NegFdbk1PosResetAfterNegOutReq';
		16#C050:
		Diag.DiagText := 'NegFdbk2AfterNegOutReq';
		16#C051:
		Diag.DiagText := 'NegFdbk2PosResetAfterNegOutReq';
		16#C060:
		Diag.DiagText := 'NegFdbk1Fdbk2AfterNegOutReq';
		16#C061:
		Diag.DiagText := 'NegFdbk1Fdbk2PosResetAfterNegOutReq';
		16#C070:
		Diag.DiagText := 'PosFdbk1AfterPosOutReq';
		16#C071:
		Diag.DiagText := 'PosFdbk1PosResetAfterPosOutReq';
		16#C080:
		Diag.DiagText := 'PosFdbk2AfterPosOutReq';
		16#C081:
		Diag.DiagText := 'PosFdbk2PosResetAfterPosOutReq';
		16#C090:
		Diag.DiagText := 'PosFdbk1Fdbk2AfterPosOutReq';
		16#C091:
		Diag.DiagText := 'PosFdbk1Fdbk2PosResetAfterPosOutReq';
		16#C111:
		Diag.DiagText := 'SameTimePosEdgeOutReqPosEdgeReset';
	END_CASE

END_ACTION
